  MoveL 660 to (60.77, 126.66, 55.41) mm, rotated rx -112.39 ry 0 rz 153.96 deg; joints [6.851, -47.635, 74.917, -1.241, 56.21, -13.391, 34.019]
  MoveL 661 to (66.75, 124.73, 52.87) mm, rotated rx -111.36 ry 0 rz 151.44 deg; joints [6.623, -47.631, 74.812, -1.242, 56.128, -12.588, 36.717]
  MoveL 662 to (67.07, 124.6, 52.75) mm, rotated rx -111.21 ry 0 rz 151.11 deg; joints [6.599, -47.654, 74.802, -1.244, 56.128, -12.462, 37.079]
  MoveL 663 to (71.33, 123.43, 49.83) mm, rotated rx -110.03 ry 0 rz 149.39 deg; joints [6.337, -47.654, 74.694, -1.241, 56.035, -11.548, 38.999]
  MoveL 664 to (71.29, 123.43, 49.87) mm, rotated rx -109.41 ry 0 rz 148.99 deg; joints [6.253, -47.698, 74.655, -1.242, 56.035, -11.007, 39.475]
  MoveL 665 to (71.98, 123.95, 47.56) mm, rotated rx -108.48 ry 0 rz 148.86 deg; joints [6.046, -47.698, 74.577, -1.235, 55.971, -10.294, 39.744]
  MoveL 666 to (72.34, 124.04, 46.77) mm, rotated rx -108.48 ry 0 rz 148.86 deg; joints [6.02, -47.694, 74.577, -1.235, 55.942, -10.32, 39.769]
  MoveL 667 to (72.46, 124.04, 46.59) mm, rotated rx -108.41 ry 0 rz 148.82 deg; joints [6.003, -47.694, 74.571, -1.234, 55.937, -10.264, 39.82]
  MoveL 668 to (72.72, 124.02, 46.25) mm, rotated rx -108.41 ry 0 rz 148.82 deg; joints [5.992, -47.687, 74.571, -1.234, 55.922, -10.276, 39.827]
  MoveL 669 to (73.92, 123.81, 44.88) mm, rotated rx -107.79 ry 0 rz 148.32 deg; joints [5.859, -47.687, 74.517, -1.226, 55.898, -9.795, 40.405]
  MoveL 670 to (74.21, 123.77, 44.51) mm, rotated rx -107.28 ry 0 rz 148.07 deg; joints [5.775, -47.695, 74.479, -1.22, 55.898, -9.373, 40.699]
  MoveL 671 to (76.55, 125.04, 36.2) mm, rotated rx -104.01 ry 0 rz 147.56 deg; joints [5.033, -47.695, 74.261, -1.159, 55.732, -6.875, 41.585]
  MoveL 672 to (76.56, 125.03, 36.23) mm, rotated rx -103.38 ry 0 rz 147.69 deg; joints [4.944, -47.695, 74.256, -1.152, 55.68, -6.332, 41.508]
  MoveL 673 to (75.15, 126.78, 32.95) mm, rotated rx -102.1 ry 0 rz 148.52 deg; joints [4.651, -47.696, 74.189, -1.119, 55.632, -5.36, 40.791]
  MoveL 674 to (75.18, 126.76, 32.96) mm, rotated rx -101.72 ry 0 rz 149 deg; joints [4.596, -47.646, 74.189, -1.111, 55.58, -5.038, 40.319]
  MoveL 675 to (72.12, 128.85, 31.65) mm, rotated rx -101.21 ry 0 rz 150.43 deg; joints [4.479, -47.646, 74.165, -1.097, 55.564, -4.653, 38.919]
  MoveL 676 to (72.16, 128.83, 31.66) mm, rotated rx -101.17 ry 0 rz 150.93 deg; joints [4.473, -47.583, 74.165, -1.092, 55.536, -4.625, 38.388]
  MoveL 677 to (69.26, 130.27, 32.26) mm, rotated rx -101.4 ry 0 rz 152.18 deg; joints [4.526, -47.583, 74.176, -1.098, 55.543, -4.801, 37.119]
  MoveL 678 to (68.73, 130.53, 32.34) mm, rotated rx -101.43 ry 0 rz 152.35 deg; joints [4.532, -47.591, 74.178, -1.1, 55.545, -4.816, 36.951]
  MoveL 679 to (65.39, 132.13, 32.76) mm, rotated rx -101.64 ry 0 rz 154.01 deg; joints [4.577, -47.56, 74.185, -1.103, 55.545, -4.988, 35.254]
  MoveL 680 to (65.13, 132.23, 32.87) mm, rotated rx -101.68 ry 0 rz 154.12 deg; joints [4.586, -47.561, 74.186, -1.104, 55.546, -5.018, 35.145]
  MoveL 681 to (65.15, 132.23, 32.84) mm, rotated rx -101.9 ry 0 rz 154.47 deg; joints [4.615, -47.509, 74.186, -1.102, 55.544, -5.211, 34.742]
  MoveL 682 to (59.71, 133.3, 38.37) mm, rotated rx -104.07 ry 0 rz 156.58 deg; joints [5.109, -47.509, 74.305, -1.155, 55.627, -6.851, 32.439]
  MoveL 683 to (58.71, 133.57, 39) mm, rotated rx -104.07 ry 0 rz 156.58 deg; joints [5.131, -47.553, 74.305, -1.16, 55.659, -6.827, 32.451]
  MoveL 684 to (58.23, 133.73, 39.16) mm, rotated rx -104.13 ry 0 rz 156.78 deg; joints [5.145, -47.553, 74.308, -1.162, 55.662, -6.875, 32.25]
  MoveL 685 to (57.76, 133.9, 39.27) mm, rotated rx -104.13 ry 0 rz 156.78 deg; joints [5.15, -47.577, 74.308, -1.164, 55.674, -6.87, 32.262]
  MoveL 686 to (52.25, 135.95, 39.92) mm, rotated rx -104.39 ry 0 rz 159.09 deg; joints [5.208, -47.577, 74.324, -1.169, 55.685, -7.065, 29.926]
  MoveL 687 to (51.7, 136.16, 39.92) mm, rotated rx -104.39 ry 0 rz 159.09 deg; joints [5.209, -47.606, 74.324, -1.172, 55.696, -7.063, 29.944]
  MoveL 688 to (50.6, 136.72, 39.43) mm, rotated rx -104.39 ry 0 rz 159.09 deg; joints [5.194, -47.671, 74.325, -1.176, 55.709, -7.076, 29.996]
  MoveL 689 to (50.38, 136.86, 39.24) mm, rotated rx -104.31 ry 0 rz 159.19 deg; joints [5.177, -47.671, 74.32, -1.175, 55.705, -7.018, 29.902]
  MoveL 690 to (49.72, 137.39, 38.2) mm, rotated rx -104.31 ry 0 rz 159.19 deg; joints [5.143, -47.715, 74.316, -1.176, 55.705, -7.052, 29.95]
  MoveL 691 to (49.04, 138.28, 35.81) mm, rotated rx -103.37 ry 0 rz 159.56 deg; joints [4.93, -47.715, 74.262, -1.154, 55.666, -6.341, 29.667]
  MoveL 692 to (48.96, 138.42, 35.38) mm, rotated rx -103.37 ry 0 rz 159.56 deg; joints [4.916, -47.721, 74.258, -1.153, 55.666, -6.356, 29.676]
  MoveL 693 to (49.06, 138.63, 34.37) mm, rotated rx -103.37 ry 0 rz 159.56 deg; joints [4.882, -47.721, 74.251, -1.15, 55.658, -6.392, 29.691]
  MoveL 694 to (49.13, 138.66, 34.16) mm, rotated rx -103.29 ry 0 rz 159.54 deg; joints [4.863, -47.721, 74.246, -1.148, 55.655, -6.331, 29.718]
  MoveL 695 to (49.47, 138.71, 33.44) mm, rotated rx -103.29 ry 0 rz 159.54 deg; joints [4.839, -47.712, 74.246, -1.145, 55.635, -6.356, 29.727]
  MoveL 696 to (50.81, 138.69, 31.45) mm, rotated rx -102.52 ry 0 rz 159.05 deg; joints [4.662, -47.712, 74.207, -1.125, 55.608, -5.771, 30.282]
  MoveL 697 to (51.64, 138.87, 29.25) mm, rotated rx -101.46 ry 0 rz 158.68 deg; joints [4.436, -47.712, 74.148, -1.094, 55.603, -4.949, 30.713]
  MoveL 698 to (51.92, 138.88, 28.69) mm, rotated rx -101.46 ry 0 rz 158.68 deg; joints [4.417, -47.702, 74.148, -1.092, 55.59, -4.969, 30.717]
  MoveL 699 to (52.11, 138.87, 28.42) mm, rotated rx -101.35 ry 0 rz 158.62 deg; joints [4.392, -47.702, 74.143, -1.089, 55.587, -4.89, 30.791]
  MoveL 700 to (52.33, 138.84, 28.13) mm, rotated rx -101.35 ry 0 rz 158.62 deg; joints [4.383, -47.694, 74.143, -1.087, 55.578, -4.9, 30.791]
  MoveL 701 to (53.88, 138.59, 26.37) mm, rotated rx -100.68 ry 0 rz 158.03 deg; joints [4.227, -47.693, 74.116, -1.066, 55.561, -4.391, 31.423]
  MoveL 702 to (53.87, 138.59, 26.41) mm, rotated rx -100.23 ry 0 rz 157.81 deg; joints [4.165, -47.724, 74.108, -1.06, 55.561, -4.012, 31.676]
  MoveL 703 to (54.09, 138.69, 25.45) mm, rotated rx -99.86 ry 0 rz 157.75 deg; joints [4.08, -47.724, 74.095, -1.048, 55.553, -3.735, 31.76]
  MoveL 704 to (54.13, 138.66, 25.45) mm, rotated rx -98.75 ry 0 rz 158.69 deg; joints [3.919, -47.625, 74.095, -1.022, 55.453, -2.799, 30.817]
  MoveL 705 to (46.69, 141.33, 25.56) mm, rotated rx -98.79 ry 0 rz 161.73 deg; joints [3.928, -47.625, 74.096, -1.023, 55.453, -2.829, 27.774]
  MoveL 706 to (46.19, 141.5, 25.51) mm, rotated rx -98.79 ry 0 rz 161.73 deg; joints [3.927, -47.651, 74.096, -1.025, 55.463, -2.83, 27.79]
  MoveL 707 to (45.76, 141.66, 25.42) mm, rotated rx -98.76 ry 0 rz 161.91 deg; joints [3.919, -47.651, 74.094, -1.024, 55.463, -2.803, 27.616]
  MoveL 708 to (44.74, 142.08, 24.9) mm, rotated rx -98.76 ry 0 rz 161.91 deg; joints [3.903, -47.707, 74.094, -1.025, 55.48, -2.819, 27.654]
  MoveL 709 to (41.28, 143.63, 21.8) mm, rotated rx -97.57 ry 0 rz 163.35 deg; joints [3.628, -47.707, 74.061, -0.983, 55.462, -1.926, 26.251]
  MoveL 710 to (40.62, 143.96, 20.83) mm, rotated rx -97.57 ry 0 rz 163.35 deg; joints [3.596, -47.745, 74.061, -0.98, 55.47, -1.959, 26.281]
  MoveL 711 to (40.51, 144.16, 19.63) mm, rotated rx -97.57 ry 0 rz 163.35 deg; joints [3.556, -47.754, 74.058, -0.975, 55.47, -2.002, 26.293]
  MoveL 712 to (40.56, 144.19, 19.26) mm, rotated rx -97.43 ry 0 rz 163.34 deg; joints [3.524, -47.754, 74.055, -0.97, 55.469, -1.897, 26.312]
  MoveL 713 to (40.77, 144.23, 18.53) mm, rotated rx -97.43 ry 0 rz 163.34 deg; joints [3.499, -47.746, 74.055, -0.965, 55.462, -1.924, 26.312]
  MoveL 714 to (42.09, 144.19, 15.65) mm, rotated rx -96.33 ry 0 rz 162.85 deg; joints [3.244, -47.746, 74.035, -0.923, 55.455, -1.102, 26.821]
  MoveL 715 to (42.15, 144.21, 15.29) mm, rotated rx -96.03 ry 0 rz 162.78 deg; joints [3.189, -47.754, 74.033, -0.915, 55.455, -0.864, 26.904]
  MoveL 716 to (43.13, 144.27, 11.53) mm, rotated rx -94.6 ry 0 rz 162.43 deg; joints [2.857, -47.755, 74.02, -0.858, 55.455, 0.205, 27.261]
  MoveL 717 to (43.15, 144.26, 11.55) mm, rotated rx -93.63 ry 0 rz 162.78 deg; joints [2.716, -47.713, 74.02, -0.831, 55.435, 1.024, 26.893]
  MoveL 718 to (37.84, 146.01, 7.35) mm, rotated rx -92.03 ry 0 rz 164.9 deg; joints [2.344, -47.713, 74.024, -0.764, 55.452, 2.216, 24.742]
  MoveL 719 to (37.83, 146.02, 7.37) mm, rotated rx -91.85 ry 0 rz 165.55 deg; joints [2.317, -47.629, 74.024, -0.755, 55.419, 2.366, 24.038]
  MoveL 720 to (29.7, 147.83, 8.53) mm, rotated rx -92.3 ry 0 rz 168.77 deg; joints [2.421, -47.626, 74.024, -0.774, 55.405, 2.032, 20.832]
  MoveL 721 to (28.41, 148.09, 8.36) mm, rotated rx -92.3 ry 0 rz 168.77 deg; joints [2.416, -47.69, 74.024, -0.776, 55.433, 2.027, 20.868]
  MoveL 722 to (28.01, 148.18, 8.19) mm, rotated rx -92.23 ry 0 rz 168.93 deg; joints [2.401, -47.69, 74.025, -0.773, 55.433, 2.076, 20.712]
  MoveL 723 to (25.31, 148.72, 6.82) mm, rotated rx -91.74 ry 0 rz 169.92 deg; joints [2.283, -47.692, 74.025, -0.752, 55.451, 2.443, 19.703]
  MoveL 724 to (25.34, 148.72, 6.79) mm, rotated rx -91.84 ry 0 rz 170.93 deg; joints [2.295, -47.562, 74.025, -0.748, 55.394, 2.352, 18.619]
  MoveL 725 to (23.1, 148.99, 8.62) mm, rotated rx -92.54 ry 0 rz 171.79 deg; joints [2.457, -47.562, 74.02, -0.778, 55.384, 1.832, 17.778]
  MoveL 726 to (22.86, 149.01, 8.97) mm, rotated rx -92.78 ry 0 rz 171.99 deg; joints [2.503, -47.549, 74.02, -0.785, 55.374, 1.64, 17.57]
  MoveL 727 to (20.3, 149.18, 11.9) mm, rotated rx -93.9 ry 0 rz 172.97 deg; joints [2.763, -47.548, 74.02, -0.831, 55.365, 0.807, 16.605]
  MoveL 728 to (19.26, 149.26, 12.61) mm, rotated rx -93.9 ry 0 rz 172.97 deg; joints [2.787, -47.599, 74.02, -0.838, 55.385, 0.834, 16.635]
  MoveL 729 to (18.7, 149.31, 12.81) mm, rotated rx -93.97 ry 0 rz 173.18 deg; joints [2.805, -47.598, 74.02, -0.841, 55.385, 0.777, 16.421]
  MoveL 730 to (18.28, 149.35, 12.92) mm, rotated rx -93.97 ry 0 rz 173.18 deg; joints [2.809, -47.619, 74.02, -0.843, 55.394, 0.782, 16.433]
  MoveL 731 to (13.22, 149.81, 13.78) mm, rotated rx -94.38 ry 0 rz 175.37 deg; joints [2.897, -47.584, 74.02, -0.856, 55.383, 0.467, 14.224]
  MoveL 732 to (10.64, 149.89, 15.02) mm, rotated rx -94.86 ry 0 rz 176.35 deg; joints [3.006, -47.583, 74.023, -0.875, 55.384, 0.114, 13.236]
  MoveL 733 to (9.93, 149.91, 15.35) mm, rotated rx -94.92 ry 0 rz 176.45 deg; joints [3.026, -47.604, 74.023, -0.879, 55.394, 0.075, 13.148]
  MoveL 734 to (7.35, 149.99, 16.03) mm, rotated rx -95.18 ry 0 rz 177.44 deg; joints [3.087, -47.604, 74.026, -0.889, 55.394, -0.119, 12.161]
  MoveL 735 to (8.24, 169.89, 17.83) mm, rotated rx -95.18 ry 0 rz 177.44 deg; joints [3.116, -46.976, 72.196, -1.011, 55.394, -0.037, 13.368]
  Set speed (1000.0 mm/s)
  MoveL 736 to (4.59, 170.21, 15.87) mm, rotated rx -94.56 ry 0 rz 178.8 deg; joints [2.963, -46.964, 72.196, -0.981, 55.377, 0.408, 12.008]
  Set speed (5.0 mm/s)
  MoveL 737 to (4.17, 150.28, 14.28) mm, rotated rx -94.56 ry 0 rz 178.8 deg; joints [2.94, -47.591, 74.026, -0.864, 55.377, 0.334, 10.801]
  Set speed (16.7 mm/s)
  MoveL 738 to (2.77, 150.26, 14.91) mm, rotated rx -94.8 ry 0 rz 179.33 deg; joints [2.995, -47.591, 74.027, -0.874, 55.377, 0.156, 10.266]
  MoveL 739 to (1.49, 150.25, 15.12) mm, rotated rx -94.8 ry 0 rz 179.33 deg; joints [3.003, -47.653, 74.027, -0.878, 55.403, 0.165, 10.302]
  MoveL 740 to (1.28, 150.26, 15.1) mm, rotated rx -94.79 ry 0 rz 179.42 deg; joints [3.001, -47.653, 74.027, -0.878, 55.403, 0.172, 10.222]
  MoveL 741 to (0.58, 150.28, 14.92) mm, rotated rx -94.79 ry 0 rz 179.42 deg; joints [2.996, -47.687, 74.027, -0.879, 55.417, 0.166, 10.242]
  MoveL 742 to (-0.95, 150.34, 14.29) mm, rotated rx -94.55 ry 0 rz 180 deg; joints [2.94, -47.687, 74.026, -0.869, 55.417, 0.344, 9.659]
  MoveL 743 to (-2.76, 150.39, 13.54) mm, rotated rx -94.27 ry 0 rz -179.31 deg; joints [2.874, -47.688, 74.024, -0.858, 55.417, 0.558, 8.969]
  MoveL 744 to (-3.05, 150.39, 13.4) mm, rotated rx -94.27 ry 0 rz -179.31 deg; joints [2.87, -47.702, 74.024, -0.858, 55.423, 0.554, 8.978]
  MoveL 745 to (-3.44, 150.4, 13.18) mm, rotated rx -94.18 ry 0 rz -179.16 deg; joints [2.85, -47.702, 74.024, -0.854, 55.423, 0.617, 8.829]
  MoveL 746 to (-5.89, 150.44, 11.76) mm, rotated rx -93.65 ry 0 rz -178.24 deg; joints [2.725, -47.705, 74.024, -0.833, 55.423, 1.017, 7.906]
  MoveL 747 to (-5.83, 150.44, 11.77) mm, rotated rx -93.52 ry 0 rz -177.74 deg; joints [2.706, -47.638, 74.024, -0.826, 55.395, 1.122, 7.365]
  MoveL 748 to (-8.98, 150.28, 11.92) mm, rotated rx -93.58 ry 0 rz -176.54 deg; joints [2.719, -47.638, 74.024, -0.828, 55.395, 1.079, 6.165]
  MoveL 749 to (-9.52, 150.25, 11.88) mm, rotated rx -93.58 ry 0 rz -176.54 deg; joints [2.718, -47.664, 74.024, -0.83, 55.406, 1.079, 6.181]
  MoveL 750 to (-10.04, 150.22, 11.79) mm, rotated rx -93.54 ry 0 rz -176.34 deg; joints [2.71, -47.664, 74.024, -0.828, 55.406, 1.105, 5.981]
  MoveL 751 to (-10.45, 150.2, 11.69) mm, rotated rx -93.54 ry 0 rz -176.34 deg; joints [2.707, -47.684, 74.024, -0.829, 55.414, 1.102, 5.993]
  MoveL 752 to (-13.43, 150.04, 10.65) mm, rotated rx -93.15 ry 0 rz -175.2 deg; joints [2.615, -47.684, 74.024, -0.812, 55.418, 1.397, 4.851]
  MoveL 753 to (-13.42, 150.04, 10.63) mm, rotated rx -93.18 ry 0 rz -174.48 deg; joints [2.618, -47.592, 74.024, -0.808, 55.379, 1.365, 4.081]
  MoveL 754 to (-16.19, 149.67, 11.96) mm, rotated rx -93.68 ry 0 rz -173.42 deg; joints [2.735, -47.592, 74.024, -0.829, 55.375, 0.99, 3.023]
  MoveL 755 to (-16.97, 149.57, 12.18) mm, rotated rx -93.68 ry 0 rz -173.42 deg; joints [2.743, -47.63, 74.024, -0.832, 55.391, 0.999, 3.046]
  MoveL 756 to (-17.85, 149.46, 12.28) mm, rotated rx -93.72 ry 0 rz -173.08 deg; joints [2.752, -47.63, 74.024, -0.834, 55.391, 0.97, 2.709]
  MoveL 757 to (-19.05, 149.32, 12.12) mm, rotated rx -93.72 ry 0 rz -173.08 deg; joints [2.748, -47.689, 74.024, -0.836, 55.416, 0.966, 2.743]
  MoveL 758 to (-23.23, 148.85, 10.44) mm, rotated rx -93.08 ry 0 rz -171.48 deg; joints [2.599, -47.689, 74.024, -0.809, 55.42, 1.444, 1.136]
  MoveL 759 to (-23.2, 148.86, 10.45) mm, rotated rx -93.07 ry 0 rz -170.84 deg; joints [2.596, -47.606, 74.024, -0.805, 55.385, 1.454, 0.451]
  MoveL 760 to (-25.12, 148.5, 11.09) mm, rotated rx -93.31 ry 0 rz -170.1 deg; joints [2.652, -47.606, 74.024, -0.815, 55.383, 1.273, -0.288]
  MoveL 761 to (-26.31, 148.29, 11.17) mm, rotated rx -93.2 ry 0 rz -170.09 deg; joints [2.64, -47.663, 74.024, -0.816, 55.407, 1.372, -0.273]
  MoveL 762 to (-27.06, 148.18, 10.9) mm, rotated rx -93.13 ry 0 rz -170.07 deg; joints [2.621, -47.698, 74.024, -0.814, 55.423, 1.425, -0.264]
  MoveL 763 to (-27.67, 148.1, 10.44) mm, rotated rx -93.06 ry 0 rz -170.06 deg; joints [2.595, -47.726, 74.024, -0.81, 55.436, 1.468, -0.261]
  MoveL 764 to (-28.2, 148.05, 9.57) mm, rotated rx -92.96 ry 0 rz -170.05 deg; joints [2.553, -47.75, 74.024, -0.804, 55.449, 1.516, -0.264]
  MoveL 765 to (-28.34, 148.09, 8.55) mm, rotated rx -92.87 ry 0 rz -170.04 deg; joints [2.506, -47.754, 74.024, -0.795, 55.454, 1.559, -0.28]
  MoveL 766 to (-29.06, 148.04, 6.92) mm, rotated rx -92.25 ry 0 rz -169.76 deg; joints [2.361, -47.755, 74.027, -0.769, 55.461, 2.023, -0.563]
  MoveL 767 to (-28.94, 148.05, 7.15) mm, rotated rx -92.25 ry 0 rz -169.76 deg; joints [2.369, -47.749, 74.027, -0.77, 55.458, 2.031, -0.566]
  MoveL 768 to (-29.05, 148.04, 6.96) mm, rotated rx -92.17 ry 0 rz -169.72 deg; joints [2.352, -47.749, 74.027, -0.767, 55.459, 2.085, -0.608]
  MoveL 769 to (-29.31, 148.01, 6.46) mm, rotated rx -92.03 ry 0 rz -169.65 deg; joints [2.314, -47.751, 74.027, -0.76, 55.465, 2.19, -0.686]
  MoveL 770 to (-29.27, 148.01, 6.49) mm, rotated rx -91.56 ry 0 rz -169.1 deg; joints [2.246, -47.676, 74.027, -0.744, 55.443, 2.584, -1.29]
  MoveL 771 to (-31.93, 147.5, 5.64) mm, rotated rx -91.23 ry 0 rz -168.07 deg; joints [2.17, -47.676, 74.03, -0.73, 55.448, 2.824, -2.327]
  MoveL 772 to (-32.39, 147.41, 5.43) mm, rotated rx -91.23 ry 0 rz -168.07 deg; joints [2.164, -47.699, 74.03, -0.73, 55.459, 2.817, -2.315]
  MoveL 773 to (-32.76, 147.33, 5.22) mm, rotated rx -91.15 ry 0 rz -167.93 deg; joints [2.145, -47.699, 74.032, -0.727, 55.46, 2.877, -2.462]
  MoveL 774 to (-33.25, 147.24, 4.86) mm, rotated rx -91.15 ry 0 rz -167.93 deg; joints [2.134, -47.722, 74.032, -0.725, 55.472, 2.864, -2.45]
  MoveL 775 to (-36.36, 146.57, 1.84) mm, rotated rx -90.01 ry 0 rz -166.72 deg; joints [1.867, -47.722, 74.049, -0.676, 55.497, 3.717, -3.706]
  MoveL 776 to (-36.4, 146.55, 1.78) mm, rotated rx -89.81 ry 0 rz -166.43 deg; joints [1.835, -47.684, 74.049, -0.668, 55.491, 3.884, -4.024]
  MoveL 777 to (-41.32, 145.25, -0.45) mm, rotated rx -88.96 ry 0 rz -164.5 deg; joints [1.638, -47.685, 74.067, -0.631, 55.513, 4.515, -5.996]
  MoveL 778 to (-41.25, 145.28, -0.43) mm, rotated rx -88.89 ry 0 rz -164.17 deg; joints [1.628, -47.637, 74.067, -0.627, 55.497, 4.575, -6.361]
  MoveL 779 to (-45.56, 143.99, -0.15) mm, rotated rx -89 ry 0 rz -162.38 deg; joints [1.653, -47.63, 74.067, -0.632, 55.485, 4.493, -8.142]
  MoveL 780 to (-46.02, 143.84, -0.16) mm, rotated rx -89 ry 0 rz -162.38 deg; joints [1.653, -47.653, 74.067, -0.633, 55.495, 4.493, -8.128]
  MoveL 781 to (-47.03, 143.51, -0.3) mm, rotated rx -88.95 ry 0 rz -161.98 deg; joints [1.641, -47.653, 74.069, -0.631, 55.496, 4.532, -8.537]
  MoveL 782 to (-47.66, 143.3, -0.48) mm, rotated rx -88.95 ry 0 rz -161.98 deg; joints [1.635, -47.685, 74.069, -0.631, 55.511, 4.527, -8.52]
  MoveL 783 to (-54.7, 140.72, -3.71) mm, rotated rx -87.72 ry 0 rz -159.13 deg; joints [1.35, -47.685, 74.103, -0.577, 55.55, 5.44, -11.441]
  MoveL 784 to (-54.97, 140.61, -3.86) mm, rotated rx -87.72 ry 0 rz -159.13 deg; joints [1.345, -47.698, 74.103, -0.577, 55.558, 5.435, -11.435]
  MoveL 785 to (-55.36, 140.45, -4.11) mm, rotated rx -87.62 ry 0 rz -158.97 deg; joints [1.323, -47.698, 74.106, -0.572, 55.561, 5.507, -11.604]
  MoveL 786 to (-55.65, 140.33, -4.33) mm, rotated rx -87.62 ry 0 rz -158.97 deg; joints [1.316, -47.712, 74.106, -0.571, 55.57, 5.499, -11.599]
  MoveL 787 to (-58.19, 139.2, -6.59) mm, rotated rx -86.76 ry 0 rz -157.91 deg; joints [1.116, -47.712, 74.136, -0.534, 55.601, 6.141, -12.718]
  MoveL 788 to (-58.87, 138.86, -7.66) mm, rotated rx -86.76 ry 0 rz -157.91 deg; joints [1.081, -47.743, 74.136, -0.528, 55.632, 6.102, -12.717]
  MoveL 789 to (-58.95, 138.82, -7.88) mm, rotated rx -86.68 ry 0 rz -157.88 deg; joints [1.061, -47.744, 74.139, -0.524, 55.636, 6.166, -12.756]
  MoveL 790 to (-59.04, 138.76, -8.27) mm, rotated rx -86.68 ry 0 rz -157.88 deg; joints [1.048, -47.748, 74.14, -0.522, 55.642, 6.152, -12.76]
  MoveL 791 to (-59.34, 138.5, -10.19) mm, rotated rx -85.95 ry 0 rz -157.74 deg; joints [0.879, -47.748, 74.17, -0.49, 55.673, 6.695, -12.965]
  MoveL 792 to (-59.48, 138.42, -10.44) mm, rotated rx -85.61 ry 0 rz -157.6 deg; joints [0.822, -47.741, 74.185, -0.479, 55.673, 6.968, -13.13]
  MoveL 793 to (-61.44, 137.13, -15.06) mm, rotated rx -83.86 ry 0 rz -156.72 deg; joints [0.415, -47.741, 74.272, -0.404, 55.76, 8.281, -14.185]
  MoveL 794 to (-61.42, 137.14, -15.03) mm, rotated rx -83.46 ry 0 rz -156.34 deg; joints [0.358, -47.687, 74.281, -0.392, 55.76, 8.616, -14.629]
  MoveL 795 to (-63.42, 136.09, -16.28) mm, rotated rx -82.98 ry 0 rz -155.48 deg; joints [0.248, -47.687, 74.308, -0.373, 55.787, 8.972, -15.545]
  MoveL 796 to (-63.67, 135.95, -16.43) mm, rotated rx -82.92 ry 0 rz -155.36 deg; joints [0.234, -47.687, 74.312, -0.37, 55.788, 9.019, -15.667]
  MoveL 797 to (-65.55, 134.9, -17.63) mm, rotated rx -82.47 ry 0 rz -154.55 deg; joints [0.129, -47.687, 74.338, -0.351, 55.818, 9.356, -16.532]
  MoveL 798 to (-65.54, 134.91, -17.62) mm, rotated rx -82.36 ry 0 rz -154.01 deg; joints [0.113, -47.612, 74.338, -0.347, 55.802, 9.45, -17.132]
  MoveL 799 to (-66.71, 134.35, -17.51) mm, rotated rx -82.4 ry 0 rz -153.51 deg; joints [0.122, -47.612, 74.336, -0.349, 55.799, 9.42, -17.624]
  MoveL 800 to (-67.08, 134.17, -17.51) mm, rotated rx -82.4 ry 0 rz -153.51 deg; joints [0.123, -47.633, 74.336, -0.349, 55.807, 9.42, -17.611]
  MoveL 801 to (-67.61, 133.9, -17.56) mm, rotated rx -82.38 ry 0 rz -153.29 deg; joints [0.118, -47.633, 74.337, -0.348, 55.808, 9.434, -17.837]
  MoveL 802 to (-67.99, 133.69, -17.63) mm, rotated rx -82.38 ry 0 rz -153.29 deg; joints [0.116, -47.654, 74.337, -0.348, 55.818, 9.431, -17.826]
  MoveL 803 to (-71.95, 131.43, -18.84) mm, rotated rx -81.92 ry 0 rz -151.55 deg; joints [0.01, -47.654, 74.366, -0.329, 55.846, 9.777, -19.625]
  MoveL 804 to (-72.27, 131.25, -18.94) mm, rotated rx -81.88 ry 0 rz -151.42 deg; joints [0.001, -47.654, 74.367, -0.328, 55.852, 9.803, -19.759]
  MoveL 805 to (-74.67, 129.78, -19.68) mm, rotated rx -81.6 ry 0 rz -150.33 deg; joints [-0.064, -47.654, 74.387, -0.317, 55.866, 10.017, -20.886]
  MoveL 806 to (-75.35, 129.33, -20.05) mm, rotated rx -81.6 ry 0 rz -150.33 deg; joints [-0.077, -47.69, 74.387, -0.315, 55.89, 10.004, -20.874]
  MoveL 807 to (-75.55, 129.19, -20.23) mm, rotated rx -81.53 ry 0 rz -150.23 deg; joints [-0.092, -47.69, 74.392, -0.312, 55.894, 10.054, -20.977]
  MoveL 808 to (-75.96, 128.88, -20.7) mm, rotated rx -81.53 ry 0 rz -150.23 deg; joints [-0.108, -47.71, 74.392, -0.31, 55.916, 10.037, -20.979]
  MoveL 809 to (-76.86, 128.09, -22.15) mm, rotated rx -80.97 ry 0 rz -149.79 deg; joints [-0.236, -47.71, 74.43, -0.288, 55.953, 10.454, -21.503]
  MoveL 810 to (-76.83, 128.11, -22.14) mm, rotated rx -80.62 ry 0 rz -149.03 deg; joints [-0.286, -47.598, 74.432, -0.277, 55.953, 10.75, -22.374]
  MoveL 811 to (-78.76, 126.95, -22.09) mm, rotated rx -80.64 ry 0 rz -148.16 deg; joints [-0.282, -47.598, 74.431, -0.278, 55.952, 10.737, -23.238]
  MoveL 812 to (-79.07, 126.75, -22.11) mm, rotated rx -80.64 ry 0 rz -148.16 deg; joints [-0.282, -47.616, 74.431, -0.278, 55.959, 10.736, -23.227]
  MoveL 813 to (-79.56, 126.43, -22.19) mm, rotated rx -80.61 ry 0 rz -147.94 deg; joints [-0.289, -47.616, 74.433, -0.277, 55.961, 10.757, -23.456]
  MoveL 814 to (-83.97, 123.36, -23.2) mm, rotated rx -80.21 ry 0 rz -145.74 deg; joints [-0.38, -47.611, 74.475, -0.262, 55.96, 11.058, -25.702]
  MoveL 815 to (-84.11, 123.27, -23.2) mm, rotated rx -80.21 ry 0 rz -145.68 deg; joints [-0.38, -47.611, 74.475, -0.262, 55.96, 11.057, -25.766]
  MoveL 816 to (-86.01, 122, -22.94) mm, rotated rx -80.32 ry 0 rz -144.71 deg; joints [-0.356, -47.607, 74.474, -0.266, 55.936, 10.978, -26.71]
  MoveL 817 to (-86.54, 121.62, -22.95) mm, rotated rx -80.32 ry 0 rz -144.71 deg; joints [-0.356, -47.639, 74.475, -0.266, 55.948, 10.977, -26.689]
  MoveL 818 to (-87.53, 120.87, -23.14) mm, rotated rx -80.25 ry 0 rz -144.23 deg; joints [-0.372, -47.639, 74.48, -0.264, 55.953, 11.031, -27.177]
  MoveL 819 to (-88.19, 120.34, -23.43) mm, rotated rx -80.25 ry 0 rz -144.23 deg; joints [-0.382, -47.678, 74.48, -0.263, 55.977, 11.021, -27.162]
  MoveL 820 to (-91.78, 117.05, -26.1) mm, rotated rx -79.22 ry 0 rz -142.37 deg; joints [-0.618, -47.678, 74.559, -0.224, 56.054, 11.794, -29.18]
  MoveL 821 to (-94.95, 113.9, -28.59) mm, rotated rx -78.17 ry 0 rz -140.41 deg; joints [-0.85, -47.678, 74.674, -0.187, 56.07, 12.597, -31.272]
  MoveL 822 to (-97.63, 111.54, -28.88) mm, rotated rx -78.03 ry 0 rz -138.89 deg; joints [-0.879, -47.662, 74.687, -0.183, 56.07, 12.701, -32.826]
  MoveL 823 to (-98.35, 110.83, -29.18) mm, rotated rx -78.03 ry 0 rz -138.89 deg; joints [-0.889, -47.709, 74.687, -0.181, 56.097, 12.691, -32.807]
  MoveL 824 to (-98.66, 110.49, -29.43) mm, rotated rx -77.93 ry 0 rz -138.71 deg; joints [-0.911, -47.709, 74.695, -0.178, 56.105, 12.764, -33]
  MoveL 825 to (-98.92, 110.18, -29.71) mm, rotated rx -77.93 ry 0 rz -138.71 deg; joints [-0.92, -47.725, 74.695, -0.177, 56.121, 12.754, -33]
  MoveL 826 to (-99.3, 109.59, -30.59) mm, rotated rx -77.93 ry 0 rz -138.71 deg; joints [-0.949, -47.747, 74.695, -0.172, 56.162, 12.722, -33.02]
  MoveL 827 to (-100.29, 106.94, -36.23) mm, rotated rx -75.74 ry 0 rz -137.74 deg; joints [-1.447, -47.748, 74.899, -0.099, 56.361, 14.379, -34.396]
  MoveL 828 to (-100.26, 106.61, -37.26) mm, rotated rx -75.74 ry 0 rz -137.74 deg; joints [-1.481, -47.748, 74.904, -0.095, 56.395, 14.343, -34.436]
  MoveL 829 to (-99.99, 106.37, -38.65) mm, rotated rx -75.2 ry 0 rz -137.75 deg; joints [-1.604, -47.748, 74.96, -0.078, 56.448, 14.755, -34.527]
  MoveL 830 to (-99.85, 106.32, -39.13) mm, rotated rx -75.2 ry 0 rz -137.75 deg; joints [-1.62, -47.748, 74.97, -0.076, 56.449, 14.738, -34.538]
  MoveL 831 to (-99.3, 106.47, -40.12) mm, rotated rx -75.2 ry 0 rz -137.75 deg; joints [-1.653, -47.727, 74.989, -0.072, 56.449, 14.703, -34.579]
  MoveL 832 to (-95.86, 107.97, -44.27) mm, rotated rx -73.55 ry 0 rz -139.17 deg; joints [-2.022, -47.727, 75.167, -0.027, 56.625, 15.957, -33.519]
  MoveL 833 to (-92.33, 109.27, -48.4) mm, rotated rx -71.91 ry 0 rz -140.58 deg; joints [-2.388, -47.727, 75.357, 0.011, 56.818, 17.217, -32.489]
  MoveL 834 to (-90.69, 109.58, -50.75) mm, rotated rx -70.84 ry 0 rz -141.26 deg; joints [-2.614, -47.727, 75.471, 0.031, 56.967, 18.047, -32.076]
  MoveL 835 to (-90.15, 109.74, -51.35) mm, rotated rx -70.54 ry 0 rz -141.5 deg; joints [-2.676, -47.727, 75.502, 0.036, 57.012, 18.285, -31.907]
  MoveL 836 to (-87.46, 109.87, -55.55) mm, rotated rx -68.83 ry 0 rz -142.4 deg; joints [-3.05, -47.727, 75.725, 0.062, 57.245, 19.606, -31.468]
  MoveL 837 to (-87.46, 109.88, -55.52) mm, rotated rx -68.22 ry 0 rz -142.48 deg; joints [-3.132, -47.727, 75.767, 0.066, 57.319, 20.135, -31.504]
  MoveL 838 to (-87.35, 108.92, -57.57) mm, rotated rx -67.38 ry 0 rz -142.27 deg; joints [-3.314, -47.727, 75.882, 0.075, 57.442, 20.786, -31.946]
  MoveL 839 to (-87.26, 108.71, -58.1) mm, rotated rx -67.38 ry 0 rz -142.27 deg; joints [-3.332, -47.727, 75.891, 0.075, 57.461, 20.768, -31.973]
  MoveL 840 to (-87.16, 108.58, -58.48) mm, rotated rx -67.22 ry 0 rz -142.27 deg; joints [-3.366, -47.727, 75.913, 0.077, 57.485, 20.892, -32.018]
  MoveL 841 to (-87.08, 108.51, -58.74) mm, rotated rx -67.22 ry 0 rz -142.27 deg; joints [-3.375, -47.727, 75.92, 0.077, 57.489, 20.883, -32.029]
  MoveL 842 to (-85.74, 107.56, -62.34) mm, rotated rx -65.73 ry 0 rz -142.48 deg; joints [-3.696, -47.727, 76.137, 0.085, 57.725, 22.05, -32.279]
  MoveL 843 to (-85.5, 107.47, -62.83) mm, rotated rx -65.73 ry 0 rz -142.48 deg; joints [-3.712, -47.727, 76.154, 0.086, 57.725, 22.034, -32.297]
  MoveL 844 to (-85.36, 107.44, -63.08) mm, rotated rx -65.63 ry 0 rz -142.52 deg; joints [-3.734, -47.727, 76.17, 0.086, 57.742, 22.115, -32.289]
  MoveL 845 to (-85.15, 107.42, -63.39) mm, rotated rx -65.63 ry 0 rz -142.52 deg; joints [-3.745, -47.723, 76.181, 0.086, 57.742, 22.105, -32.304]
  MoveL 846 to (-84.01, 107.4, -64.91) mm, rotated rx -64.99 ry 0 rz -142.89 deg; joints [-3.881, -47.723, 76.277, 0.087, 57.851, 22.609, -32.133]
  MoveL 847 to (-84.04, 107.41, -64.86) mm, rotated rx -64.47 ry 0 rz -143.01 deg; joints [-3.948, -47.723, 76.311, 0.086, 57.932, 23.059, -32.133]
  MoveL 848 to (-83.77, 106.83, -66.17) mm, rotated rx -63.92 ry 0 rz -142.95 deg; joints [-4.065, -47.735, 76.408, 0.086, 58.007, 23.492, -32.351]
  MoveL 849 to (-83.49, 106.57, -66.94) mm, rotated rx -63.92 ry 0 rz -142.95 deg; joints [-4.091, -47.736, 76.431, 0.085, 58.022, 23.467, -32.388]
  MoveL 850 to (-83.37, 106.52, -67.16) mm, rotated rx -63.82 ry 0 rz -142.98 deg; joints [-4.111, -47.739, 76.449, 0.085, 58.034, 23.542, -32.388]
  MoveL 851 to (-82.97, 106.45, -67.77) mm, rotated rx -63.82 ry 0 rz -142.98 deg; joints [-4.131, -47.732, 76.472, 0.085, 58.034, 23.522, -32.418]
  MoveL 852 to (-80.87, 106.44, -70.28) mm, rotated rx -62.75 ry 0 rz -143.69 deg; joints [-4.357, -47.732, 76.643, 0.078, 58.232, 24.374, -32.068]
  MoveL 853 to (-80.38, 106.41, -70.87) mm, rotated rx -62.47 ry 0 rz -143.87 deg; joints [-4.413, -47.732, 76.685, 0.076, 58.287, 24.596, -31.99]
  MoveL 854 to (-80.11, 106.42, -71.17) mm, rotated rx -62.47 ry 0 rz -143.87 deg; joints [-4.423, -47.725, 76.697, 0.075, 58.287, 24.586, -32.009]
  MoveL 855 to (-75.14, 106.77, -75.91) mm, rotated rx -60.41 ry 0 rz -145.73 deg; joints [-4.85, -47.725, 77.041, 0.047, 58.702, 26.239, -30.913]
  MoveL 856 to (-74.77, 106.81, -76.21) mm, rotated rx -60.41 ry 0 rz -145.73 deg; joints [-4.86, -47.711, 77.054, 0.046, 58.702, 26.229, -30.94]
  MoveL 857 to (-73.82, 107.15, -76.66) mm, rotated rx -60.41 ry 0 rz -145.73 deg; joints [-4.875, -47.665, 77.073, 0.042, 58.702, 26.217, -31.006]
  MoveL 858 to (-73.35, 107.38, -76.79) mm, rotated rx -60.35 ry 0 rz -145.96 deg; joints [-4.887, -47.665, 77.083, 0.041, 58.714, 26.261, -30.796]
  MoveL 859 to (-73.05, 107.55, -76.85) mm, rotated rx -60.35 ry 0 rz -145.96 deg; joints [-4.888, -47.647, 77.085, 0.04, 58.714, 26.26, -30.816]
  MoveL 860 to (-68.65, 110, -77.42) mm, rotated rx -60.1 ry 0 rz -148.18 deg; joints [-4.94, -47.647, 77.128, 0.035, 58.768, 26.462, -28.695]
  MoveL 861 to (-66.58, 110.63, -78.32) mm, rotated rx -59.61 ry 0 rz -149.45 deg; joints [-5.033, -47.647, 77.167, 0.022, 58.946, 26.868, -27.637]
  MoveL 862 to (-65.98, 110.84, -78.54) mm, rotated rx -59.42 ry 0 rz -149.91 deg; joints [-5.064, -47.647, 77.173, 0.018, 59.02, 27.031, -27.263]
  MoveL 863 to (-60.49, 111.53, -81.89) mm, rotated rx -57.91 ry 0 rz -152.21 deg; joints [-5.368, -47.647, 77.44, -0.021, 59.364, 28.252, -25.566]
  MoveL 864 to (-60.48, 111.53, -81.9) mm, rotated rx -57.06 ry 0 rz -152.65 deg; joints [-5.474, -47.647, 77.486, -0.041, 59.587, 29.008, -25.397]
  MoveL 865 to (-59.61, 108.8, -86.12) mm, rotated rx -55.14 ry 0 rz -152.43 deg; joints [-5.862, -47.915, 78.097, -0.067, 59.588, 30.558, -25.966]
  MoveL 866 to (-59.48, 108.55, -86.53) mm, rotated rx -55.14 ry 0 rz -152.43 deg; joints [-5.876, -47.925, 78.12, -0.068, 59.588, 30.544, -25.979]
  MoveL 867 to (-58.88, 108.18, -87.39) mm, rotated rx -55.14 ry 0 rz -152.43 deg; joints [-5.906, -47.926, 78.169, -0.072, 59.588, 30.516, -26.028]
  MoveL 868 to (-58.7, 108.13, -87.58) mm, rotated rx -55.05 ry 0 rz -152.49 deg; joints [-5.923, -47.926, 78.185, -0.075, 59.611, 30.588, -26.001]
  MoveL 869 to (-58.54, 108.09, -87.73) mm, rotated rx -55.05 ry 0 rz -152.49 deg; joints [-5.928, -47.923, 78.194, -0.076, 59.611, 30.583, -26.013]
  MoveL 870 to (-56.56, 107.72, -89.47) mm, rotated rx -54.23 ry 0 rz -153.24 deg; joints [-6.087, -47.923, 78.349, -0.11, 59.828, 31.259, -25.639]
  MoveL 871 to (-54.65, 107.13, -91.35) mm, rotated rx -53.27 ry 0 rz -153.99 deg; joints [-6.267, -47.924, 78.522, -0.153, 60.097, 32.061, -25.338]
  MoveL 872 to (-54.31, 107.05, -91.64) mm, rotated rx -53.27 ry 0 rz -153.99 deg; joints [-6.277, -47.916, 78.541, -0.156, 60.097, 32.052, -25.364]
  MoveL 873 to (-53.99, 107.01, -91.88) mm, rotated rx -53.16 ry 0 rz -154.11 deg; joints [-6.299, -47.917, 78.563, -0.161, 60.129, 32.147, -25.289]
  MoveL 874 to (-51.7, 106.68, -93.55) mm, rotated rx -52.36 ry 0 rz -155.04 deg; joints [-6.452, -47.918, 78.721, -0.202, 60.357, 32.815, -24.755]
  MoveL 875 to (-51.72, 106.71, -93.51) mm, rotated rx -51.87 ry 0 rz -155.33 deg; joints [-6.508, -47.918, 78.746, -0.22, 60.508, 33.259, -24.633]
  MoveL 876 to (-51.32, 106.17, -94.35) mm, rotated rx -51.46 ry 0 rz -155.41 deg; joints [-6.586, -47.983, 78.888, -0.23, 60.508, 33.59, -24.637]
  MoveL 877 to (-51.01, 105.9, -94.82) mm, rotated rx -51.46 ry 0 rz -155.41 deg; joints [-6.603, -47.988, 78.918, -0.233, 60.508, 33.575, -24.663]
  MoveL 878 to (-50.61, 105.7, -95.25) mm, rotated rx -51.43 ry 0 rz -155.42 deg; joints [-6.622, -47.991, 78.955, -0.237, 60.508, 33.592, -24.679]
  MoveL 879 to (-49.82, 105.45, -95.95) mm, rotated rx -51.09 ry 0 rz -155.73 deg; joints [-6.686, -47.994, 79.026, -0.256, 60.607, 33.881, -24.546]
  MoveL 880 to (-49.34, 104.96, -96.73) mm, rotated rx -50.4 ry 0 rz -156.02 deg; joints [-6.797, -48.108, 79.229, -0.269, 60.609, 34.465, -24.345]
  MoveL 881 to (-49.02, 104.73, -97.14) mm, rotated rx -50.4 ry 0 rz -156.02 deg; joints [-6.811, -48.11, 79.257, -0.273, 60.609, 34.453, -24.371]
  MoveL 882 to (-48.71, 104.57, -97.47) mm, rotated rx -50.23 ry 0 rz -156.13 deg; joints [-6.843, -48.137, 79.316, -0.277, 60.611, 34.588, -24.294]
  MoveL 883 to (-48.28, 104.42, -97.85) mm, rotated rx -50.23 ry 0 rz -156.13 deg; joints [-6.856, -48.131, 79.342, -0.281, 60.611, 34.577, -24.327]
  MoveL 884 to (-43.98, 103.32, -100.99) mm, rotated rx -48.64 ry 0 rz -157.91 deg; joints [-7.157, -48.408, 79.924, -0.327, 60.611, 35.893, -22.851]
  MoveL 885 to (-43.55, 103.24, -101.26) mm, rotated rx -48.64 ry 0 rz -157.91 deg; joints [-7.166, -48.397, 79.945, -0.331, 60.611, 35.885, -22.883]
  MoveL 886 to (-42.45, 103.34, -101.62) mm, rotated rx -48.64 ry 0 rz -157.91 deg; joints [-7.179, -48.352, 79.975, -0.34, 60.611, 35.878, -22.959]
  MoveL 887 to (-41.64, 103.55, -101.74) mm, rotated rx -48.58 ry 0 rz -158.34 deg; joints [-7.19, -48.363, 79.998, -0.342, 60.612, 35.93, -22.548]
  MoveL 888 to (-40.85, 103.85, -101.76) mm, rotated rx -48.58 ry 0 rz -158.34 deg; joints [-7.19, -48.318, 80.003, -0.348, 60.612, 35.933, -22.598]
  MoveL 889 to (-39.94, 104.31, -101.64) mm, rotated rx -48.64 ry 0 rz -158.86 deg; joints [-7.179, -48.307, 79.982, -0.346, 60.612, 35.885, -22.065]
  MoveL 890 to (-39.97, 104.32, -101.62) mm, rotated rx -47.2 ry 0 rz -160.12 deg; joints [-7.348, -48.601, 80.305, -0.357, 60.612, 37.156, -20.832]
  MoveL 891 to (-40.46, 103.11, -102.66) mm, rotated rx -46.67 ry 0 rz -159.67 deg; joints [-7.447, -48.699, 80.507, -0.374, 60.613, 37.597, -21.386]
  MoveL 892 to (-40.5, 102.15, -103.6) mm, rotated rx -46.67 ry 0 rz -159.67 deg; joints [-7.481, -48.753, 80.575, -0.378, 60.613, 37.564, -21.401]
  MoveL 893 to (-40.38, 101.81, -103.97) mm, rotated rx -46.47 ry 0 rz -159.67 deg; joints [-7.518, -48.789, 80.651, -0.384, 60.613, 37.728, -21.443]
  MoveL 894 to (-39.8, 101.13, -104.86) mm, rotated rx -46.47 ry 0 rz -159.67 deg; joints [-7.55, -48.805, 80.719, -0.392, 60.613, 37.7, -21.496]
  MoveL 895 to (-37.19, 99.47, -107.37) mm, rotated rx -45.13 ry 0 rz -160.69 deg; joints [-7.796, -49.061, 81.241, -0.438, 60.613, 38.826, -20.748]
  MoveL 896 to (-36.15, 99.14, -108.04) mm, rotated rx -45.13 ry 0 rz -160.69 deg; joints [-7.819, -49.041, 81.298, -0.45, 60.613, 38.809, -20.826]
  MoveL 897 to (-35.88, 99.12, -108.15) mm, rotated rx -45.07 ry 0 rz -160.82 deg; joints [-7.83, -49.053, 81.322, -0.452, 60.613, 38.859, -20.704]
  MoveL 898 to (-35.2, 99.14, -108.35) mm, rotated rx -45.07 ry 0 rz -160.82 deg; joints [-7.837, -49.026, 81.341, -0.458, 60.613, 38.856, -20.751]
  MoveL 899 to (-31.81, 99.55, -109.02) mm, rotated rx -44.7 ry 0 rz -162.65 deg; joints [-7.903, -49.097, 81.486, -0.471, 60.613, 39.162, -18.994]
  MoveL 900 to (-31.5, 99.6, -109.07) mm, rotated rx -44.7 ry 0 rz -162.65 deg; joints [-7.905, -49.082, 81.491, -0.474, 60.613, 39.162, -19.014]
  MoveL 901 to (-31.19, 99.66, -109.1) mm, rotated rx -44.68 ry 0 rz -162.83 deg; joints [-7.908, -49.086, 81.498, -0.475, 60.614, 39.177, -18.846]
  MoveL 902 to (-29.78, 99.83, -109.33) mm, rotated rx -44.54 ry 0 rz -163.7 deg; joints [-7.933, -49.123, 81.551, -0.478, 60.614, 39.296, -17.991]
  MoveL 903 to (-29.79, 99.83, -109.32) mm, rotated rx -43.61 ry 0 rz -164.76 deg; joints [-8.039, -49.342, 81.774, -0.485, 60.614, 40.128, -16.934]
  MoveL 904 to (-29.36, 98.21, -110.91) mm, rotated rx -42.73 ry 0 rz -164.75 deg; joints [-8.196, -49.518, 82.125, -0.519, 60.614, 40.865, -17.118]
  MoveL 905 to (-29.24, 97.91, -111.2) mm, rotated rx -42.73 ry 0 rz -164.75 deg; joints [-8.206, -49.529, 82.15, -0.521, 60.614, 40.856, -17.133]
  MoveL 906 to (-28.73, 97.35, -111.82) mm, rotated rx -42.73 ry 0 rz -164.75 deg; joints [-8.229, -49.537, 82.206, -0.529, 60.614, 40.837, -17.18]
  MoveL 907 to (-28.33, 97.08, -112.16) mm, rotated rx -42.54 ry 0 rz -164.93 deg; joints [-8.263, -49.576, 82.282, -0.536, 60.614, 40.997, -17.043]
  MoveL 908 to (-31.85, 110.14, -126.89) mm, rotated rx -42.54 ry 0 rz -164.93 deg; joints [-8.723, -48.908, 80.918, -0.467, 60.614, 40.498, -16.346]
  Set speed (1000.0 mm/s)
  MoveL 909 to (-30.55, 107.92, -129.11) mm, rotated rx -41.19 ry 0 rz -165.43 deg; joints [-8.955, -49.192, 81.459, -0.518, 60.614, 41.648, -16.105]
  Set speed (5.0 mm/s)
  MoveL 910 to (-27.24, 95.17, -114.05) mm, rotated rx -41.19 ry 0 rz -165.43 deg; joints [-8.483, -49.853, 82.794, -0.584, 60.614, 42.157, -16.779]
  Set speed (16.7 mm/s)
  MoveL 911 to (-27.07, 94.92, -114.3) mm, rotated rx -41.04 ry 0 rz -165.49 deg; joints [-8.508, -49.884, 82.855, -0.59, 60.614, 42.281, -16.752]
  MoveL 912 to (-26.62, 94.47, -114.78) mm, rotated rx -41.04 ry 0 rz -165.49 deg; joints [-8.526, -49.889, 82.9, -0.597, 60.614, 42.267, -16.792]
  MoveL 913 to (-25.14, 93.4, -115.97) mm, rotated rx -40.33 ry 0 rz -166.19 deg; joints [-8.648, -50.042, 83.194, -0.626, 60.615, 42.87, -16.239]
  MoveL 914 to (-25.15, 93.43, -115.95) mm, rotated rx -39.74 ry 0 rz -166.41 deg; joints [-8.711, -50.14, 83.344, -0.638, 60.615, 43.405, -16.07]
  MoveL 915 to (-25.01, 92.14, -117.01) mm, rotated rx -39.11 ry 0 rz -166.31 deg; joints [-8.819, -50.278, 83.609, -0.665, 60.615, 43.942, -16.296]
  MoveL 916 to (-24.75, 91.45, -117.61) mm, rotated rx -39.11 ry 0 rz -166.31 deg; joints [-8.841, -50.304, 83.667, -0.672, 60.615, 43.923, -16.328]
  MoveL 917 to (-24.52, 91.12, -117.91) mm, rotated rx -38.93 ry 0 rz -166.4 deg; joints [-8.873, -50.345, 83.745, -0.68, 60.615, 44.081, -16.281]
  MoveL 918 to (-24, 90.62, -118.4) mm, rotated rx -38.93 ry 0 rz -166.4 deg; joints [-8.891, -50.349, 83.795, -0.688, 60.615, 44.067, -16.327]
  MoveL 919 to (-22.5, 89.61, -119.46) mm, rotated rx -38.27 ry 0 rz -167.16 deg; joints [-9.001, -50.497, 84.074, -0.717, 60.615, 44.629, -15.692]
  MoveL 920 to (-22.5, 89.65, -119.43) mm, rotated rx -37.03 ry 0 rz -166.95 deg; joints [-9.129, -50.653, 84.407, -0.755, 60.615, 45.765, -16.089]
  MoveL 921 to (-24.87, 86.81, -121.05) mm, rotated rx -36.02 ry 0 rz -165.09 deg; joints [-9.295, -50.889, 84.844, -0.801, 60.615, 46.63, -18.149]
  MoveL 922 to (-25.28, 85.96, -121.57) mm, rotated rx -36.02 ry 0 rz -165.09 deg; joints [-9.316, -50.946, 84.89, -0.803, 60.626, 46.61, -18.149]
  MoveL 923 to (-25.23, 85.07, -122.2) mm, rotated rx -36.02 ry 0 rz -165.09 deg; joints [-9.341, -50.991, 84.956, -0.809, 60.626, 46.588, -18.169]
  MoveL 924 to (-25.12, 84.72, -122.47) mm, rotated rx -35.85 ry 0 rz -165.11 deg; joints [-9.37, -51.033, 85.033, -0.817, 60.626, 46.739, -18.191]
  MoveL 925 to (-24.62, 83.97, -123.09) mm, rotated rx -35.85 ry 0 rz -165.11 deg; joints [-9.394, -51.053, 85.101, -0.827, 60.626, 46.72, -18.239]
  MoveL 926 to (-22.9, 82.39, -124.47) mm, rotated rx -34.92 ry 0 rz -165.95 deg; joints [-9.543, -51.276, 85.509, -0.871, 60.626, 47.525, -17.586]
  MoveL 927 to (-22.92, 82.41, -124.46) mm, rotated rx -34.46 ry 0 rz -166.13 deg; joints [-9.588, -51.358, 85.631, -0.882, 60.626, 47.942, -17.446]
  MoveL 928 to (-22.74, 81.54, -125.06) mm, rotated rx -34.05 ry 0 rz -166.11 deg; joints [-9.653, -51.458, 85.813, -0.901, 60.626, 48.296, -17.553]
  MoveL 929 to (-22.54, 81.02, -125.44) mm, rotated rx -34.05 ry 0 rz -166.11 deg; joints [-9.668, -51.478, 85.856, -0.907, 60.626, 48.284, -17.577]
  MoveL 930 to (-22.42, 80.81, -125.59) mm, rotated rx -33.95 ry 0 rz -166.15 deg; joints [-9.685, -51.504, 85.903, -0.912, 60.626, 48.376, -17.552]
  MoveL 931 to (-22.2, 80.51, -125.83) mm, rotated rx -33.95 ry 0 rz -166.15 deg; joints [-9.694, -51.511, 85.931, -0.916, 60.626, 48.369, -17.573]
  MoveL 932 to (-21.5, 79.72, -126.44) mm, rotated rx -33.51 ry 0 rz -166.49 deg; joints [-9.762, -51.618, 86.124, -0.938, 60.626, 48.746, -17.32]
  MoveL 933 to (-21.49, 79.74, -126.44) mm, rotated rx -32.68 ry 0 rz -166.42 deg; joints [-9.843, -51.742, 86.359, -0.964, 60.626, 49.518, -17.502]
  MoveL 934 to (-22.41, 77.11, -127.9) mm, rotated rx -31.66 ry 0 rz -165.36 deg; joints [-10.001, -52.003, 86.822, -1.016, 60.626, 50.408, -18.768]
  MoveL 935 to (-22.43, 77.01, -127.96) mm, rotated rx -31.53 ry 0 rz -165.22 deg; joints [-10.015, -52.02, 86.867, -1.022, 60.626, 50.526, -18.94]
  MoveL 936 to (-23.67, 74.16, -129.41) mm, rotated rx -30.49 ry 0 rz -163.81 deg; joints [-10.173, -52.292, 87.345, -1.076, 60.626, 51.44, -20.557]
  MoveL 937 to (-23.69, 74.17, -129.4) mm, rotated rx -30.27 ry 0 rz -163.37 deg; joints [-10.193, -52.297, 87.411, -1.088, 60.626, 51.647, -21.063]
  MoveL 938 to (-26.22, 70.97, -130.7) mm, rotated rx -29.31 ry 0 rz -160.89 deg; joints [-10.336, -52.555, 87.855, -1.138, 60.626, 52.486, -23.734]
  MoveL 939 to (-29.43, 80.22, -148.14) mm, rotated rx -29.31 ry 0 rz -160.89 deg; joints [-10.903, -51.968, 86.788, -1.117, 60.626, 51.903, -23.259]
  Set speed (1000.0 mm/s)
  MoveL 940 to (-28.39, 76.79, -150.15) mm, rotated rx -29.19 ry 0 rz -160.94 deg; joints [-11.001, -52.155, 87.097, -1.151, 60.626, 51.949, -23.333]
  Set speed (5.0 mm/s)
  MoveL 941 to (-25.2, 67.57, -132.69) mm, rotated rx -29.19 ry 0 rz -160.94 deg; joints [-10.433, -52.743, 88.159, -1.171, 60.627, 52.533, -23.803]
  Set speed (16.7 mm/s)
  MoveL 942 to (-23.44, 66.82, -133.39) mm, rotated rx -28.62 ry 0 rz -162.11 deg; joints [-10.514, -52.897, 88.422, -1.2, 60.627, 53.034, -22.742]
  MoveL 943 to (-22.89, 66.66, -133.57) mm, rotated rx -28.62 ry 0 rz -162.11 deg; joints [-10.522, -52.888, 88.452, -1.208, 60.627, 53.032, -22.781]
  MoveL 944 to (-21.54, 66.75, -133.74) mm, rotated rx -28.62 ry 0 rz -162.11 deg; joints [-10.528, -52.838, 88.49, -1.225, 60.627, 53.035, -22.871]
  MoveL 945 to (-21.39, 66.8, -133.74) mm, rotated rx -28.62 ry 0 rz -162.25 deg; joints [-10.528, -52.838, 88.49, -1.225, 60.627, 53.035, -22.735]
  MoveL 946 to (-21.09, 66.94, -133.72) mm, rotated rx -28.64 ry 0 rz -162.61 deg; joints [-10.526, -52.839, 88.481, -1.223, 60.627, 53.02, -22.358]
  MoveL 947 to (-20.32, 67.13, -133.74) mm, rotated rx -28.62 ry 0 rz -163.26 deg; joints [-10.528, -52.844, 88.488, -1.224, 60.627, 53.034, -21.717]
  MoveL 948 to (-19.09, 67.49, -133.74) mm, rotated rx -28.62 ry 0 rz -164.2 deg; joints [-10.528, -52.837, 88.49, -1.225, 60.626, 53.035, -20.779]
  MoveL 949 to (-18.33, 67.84, -133.67) mm, rotated rx -28.67 ry 0 rz -164.34 deg; joints [-10.52, -52.791, 88.473, -1.229, 60.626, 52.998, -20.669]
  MoveL 950 to (-17.72, 68.39, -133.48) mm, rotated rx -28.72 ry 0 rz -164.48 deg; joints [-10.506, -52.739, 88.437, -1.23, 60.626, 52.965, -20.545]
  MoveL 951 to (-14.72, 70.88, -132.54) mm, rotated rx -29.47 ry 0 rz -167.32 deg; joints [-10.397, -52.535, 88.084, -1.19, 60.626, 52.296, -17.555]
  MoveL 952 to (-14.46, 71.1, -132.45) mm, rotated rx -29.51 ry 0 rz -167.44 deg; joints [-10.389, -52.514, 88.063, -1.189, 60.626, 52.265, -17.432]
  MoveL 953 to (-14.22, 71.35, -132.34) mm, rotated rx -29.51 ry 0 rz -167.44 deg; joints [-10.385, -52.496, 88.055, -1.188, 60.616, 52.269, -17.434]
  MoveL 954 to (-13.06, 72.66, -131.75) mm, rotated rx -29.98 ry 0 rz -168.56 deg; joints [-10.316, -52.371, 87.837, -1.163, 60.616, 51.853, -16.224]
  MoveL 955 to (-12.27, 73.21, -131.52) mm, rotated rx -30.27 ry 0 rz -169.56 deg; joints [-10.279, -52.325, 87.718, -1.146, 60.616, 51.59, -15.147]
  MoveL 956 to (-11.79, 73.66, -131.31) mm, rotated rx -30.27 ry 0 rz -169.56 deg; joints [-10.27, -52.289, 87.704, -1.146, 60.6, 51.599, -15.152]
  MoveL 957 to (-11.6, 73.89, -131.2) mm, rotated rx -30.36 ry 0 rz -169.74 deg; joints [-10.257, -52.266, 87.663, -1.141, 60.6, 51.522, -14.957]
  MoveL 958 to (-11.34, 74.28, -131) mm, rotated rx -30.36 ry 0 rz -169.74 deg; joints [-10.249, -52.237, 87.642, -1.141, 60.597, 51.531, -14.962]
  MoveL 959 to (-9.75, 77.15, -129.46) mm, rotated rx -31.52 ry 0 rz -171.29 deg; joints [-10.074, -51.933, 87.107, -1.08, 60.597, 50.505, -13.176]
  MoveL 960 to (-8.68, 78.06, -128.99) mm, rotated rx -32.08 ry 0 rz -172.54 deg; joints [-10.002, -51.835, 86.883, -1.05, 60.597, 50.001, -11.797]
  MoveL 961 to (-8.12, 78.78, -128.59) mm, rotated rx -32.08 ry 0 rz -172.54 deg; joints [-9.985, -51.78, 86.845, -1.049, 60.586, 50.018, -11.804]
  MoveL 962 to (-8.05, 78.92, -128.51) mm, rotated rx -32.14 ry 0 rz -172.6 deg; joints [-9.976, -51.764, 86.817, -1.046, 60.586, 49.965, -11.727]
  MoveL 963 to (-7.91, 79.29, -128.29) mm, rotated rx -32.14 ry 0 rz -172.6 deg; joints [-9.966, -51.74, 86.792, -1.045, 60.586, 49.974, -11.727]
  MoveL 964 to (-7.49, 80.82, -127.35) mm, rotated rx -32.81 ry 0 rz -173.04 deg; joints [-9.863, -51.57, 86.489, -1.011, 60.586, 49.388, -11.155]
  MoveL 965 to (-6.64, 82.04, -126.62) mm, rotated rx -33.57 ry 0 rz -173.96 deg; joints [-9.759, -51.419, 86.184, -0.974, 60.586, 48.711, -10.071]
  MoveL 966 to (-6.48, 82.31, -126.45) mm, rotated rx -33.57 ry 0 rz -173.96 deg; joints [-9.753, -51.4, 86.167, -0.973, 60.584, 48.718, -10.071]
  MoveL 967 to (-6.28, 82.72, -126.19) mm, rotated rx -33.75 ry 0 rz -174.14 deg; joints [-9.724, -51.355, 86.086, -0.964, 60.584, 48.559, -9.861]
  MoveL 968 to (-6.17, 82.97, -126.04) mm, rotated rx -33.75 ry 0 rz -174.14 deg; joints [-9.718, -51.339, 86.069, -0.963, 60.584, 48.565, -9.86]
  MoveL 969 to (-4.86, 86.58, -123.64) mm, rotated rx -35.38 ry 0 rz -175.25 deg; joints [-9.459, -50.942, 85.345, -0.883, 60.584, 47.15, -8.415]
  MoveL 970 to (-4.77, 87.47, -123.02) mm, rotated rx -35.38 ry 0 rz -175.25 deg; joints [-9.434, -50.897, 85.279, -0.877, 60.584, 47.172, -8.393]
  MoveL 971 to (-4.81, 87.73, -122.83) mm, rotated rx -35.51 ry 0 rz -175.23 deg; joints [-9.414, -50.867, 85.224, -0.871, 60.584, 47.064, -8.381]
  MoveL 972 to (-4.87, 87.98, -122.65) mm, rotated rx -35.51 ry 0 rz -175.23 deg; joints [-9.407, -50.859, 85.204, -0.869, 60.584, 47.07, -8.369]
  MoveL 973 to (-5.21, 89.02, -121.87) mm, rotated rx -36 ry 0 rz -175.07 deg; joints [-9.326, -50.741, 84.986, -0.845, 60.583, 46.642, -8.43]
  MoveL 974 to (-5.24, 89.01, -121.88) mm, rotated rx -36.91 ry 0 rz -175.6 deg; joints [-9.234, -50.651, 84.732, -0.81, 60.583, 45.807, -7.738]
  MoveL 975 to (-4.26, 89.78, -121.36) mm, rotated rx -37.25 ry 0 rz -176.26 deg; joints [-9.179, -50.573, 84.585, -0.794, 60.583, 45.517, -7.001]
  MoveL 976 to (-3.87, 90.15, -121.1) mm, rotated rx -37.25 ry 0 rz -176.26 deg; joints [-9.169, -50.544, 84.567, -0.794, 60.572, 45.527, -7.001]
  MoveL 977 to (-3.46, 91.17, -120.34) mm, rotated rx -37.25 ry 0 rz -176.26 deg; joints [-9.138, -50.478, 84.493, -0.79, 60.572, 45.555, -6.993]
  MoveL 978 to (-3.45, 91.36, -120.21) mm, rotated rx -37.33 ry 0 rz -176.28 deg; joints [-9.124, -50.458, 84.456, -0.786, 60.572, 45.48, -6.961]
  MoveL 979 to (-3.51, 91.87, -119.81) mm, rotated rx -37.33 ry 0 rz -176.28 deg; joints [-9.109, -50.437, 84.415, -0.781, 60.572, 45.493, -6.94]
  MoveL 980 to (-4.01, 93.64, -118.41) mm, rotated rx -38.19 ry 0 rz -176.04 deg; joints [-8.965, -50.242, 84.046, -0.742, 60.572, 44.757, -6.999]
  MoveL 981 to (-4, 93.62, -118.43) mm, rotated rx -38.58 ry 0 rz -176.07 deg; joints [-8.926, -50.191, 83.945, -0.731, 60.572, 44.407, -6.919]
  MoveL 982 to (-3.66, 94.95, -117.38) mm, rotated rx -39.22 ry 0 rz -176.33 deg; joints [-8.817, -50.048, 83.672, -0.702, 60.572, 43.858, -6.525]
  MoveL 983 to (-4.47, 107.57, -132.88) mm, rotated rx -39.22 ry 0 rz -176.33 deg; joints [-9.305, -49.394, 82.376, -0.644, 60.572, 43.336, -5.883]
  Set speed (1000.0 mm/s)
  MoveL 984 to (-3.83, 110.44, -130.52) mm, rotated rx -40.44 ry 0 rz -176.75 deg; joints [-9.085, -49.119, 81.832, -0.587, 60.572, 42.306, -5.19]
  Set speed (5.0 mm/s)
  MoveL 985 to (-3.09, 97.49, -115.3) mm, rotated rx -40.44 ry 0 rz -176.75 deg; joints [-8.607, -49.779, 83.155, -0.649, 60.571, 42.819, -5.853]
  Set speed (16.7 mm/s)
  MoveL 986 to (-2.24, 100.79, -112.45) mm, rotated rx -42.09 ry 0 rz -177.35 deg; joints [-8.32, -49.429, 82.471, -0.58, 60.571, 41.415, -4.919]
  MoveL 987 to (-2.17, 101.07, -112.19) mm, rotated rx -42.21 ry 0 rz -177.39 deg; joints [-8.297, -49.401, 82.418, -0.575, 60.571, 41.312, -4.854]
  MoveL 988 to (-1.61, 103.2, -110.24) mm, rotated rx -43.32 ry 0 rz -177.75 deg; joints [-8.102, -49.177, 81.972, -0.532, 60.571, 40.381, -4.264]
  MoveL 989 to (-1.56, 103.61, -109.86) mm, rotated rx -43.32 ry 0 rz -177.75 deg; joints [-8.088, -49.157, 81.94, -0.529, 60.571, 40.394, -4.251]
  MoveL 990 to (-1.57, 103.74, -109.74) mm, rotated rx -43.39 ry 0 rz -177.75 deg; joints [-8.075, -49.143, 81.912, -0.526, 60.571, 40.334, -4.237]
  MoveL 991 to (-1.73, 104.85, -108.68) mm, rotated rx -44.18 ry 0 rz -177.72 deg; joints [-7.948, -49.004, 81.627, -0.499, 60.571, 39.659, -4.119]
  MoveL 992 to (0.21, 108.08, -105.48) mm, rotated rx -46.08 ry 0 rz -178.91 deg; joints [-7.614, -48.657, 80.904, -0.431, 60.571, 38.047, -2.555]
  MoveL 993 to (0.42, 108.82, -104.72) mm, rotated rx -46.08 ry 0 rz -178.91 deg; joints [-7.586, -48.617, 80.846, -0.428, 60.571, 38.073, -2.538]
  MoveL 994 to (0.42, 109, -104.52) mm, rotated rx -46.19 ry 0 rz -178.9 deg; joints [-7.567, -48.598, 80.807, -0.424, 60.571, 37.987, -2.519]
  MoveL 995 to (0.32, 109.44, -104.07) mm, rotated rx -46.19 ry 0 rz -178.9 deg; joints [-7.55, -48.585, 80.772, -0.42, 60.571, 38.002, -2.496]
  MoveL 996 to (-0.31, 110.94, -102.46) mm, rotated rx -47.02 ry 0 rz -178.59 deg; joints [-7.396, -48.431, 80.452, -0.392, 60.571, 37.308, -2.638]
  MoveL 997 to (-0.3, 112.04, -101.27) mm, rotated rx -47.89 ry 0 rz -178.57 deg; joints [-7.251, -48.285, 80.159, -0.368, 60.571, 36.566, -2.518]
  MoveL 998 to (-0.34, 112.34, -100.94) mm, rotated rx -47.89 ry 0 rz -178.57 deg; joints [-7.239, -48.275, 80.135, -0.365, 60.571, 36.576, -2.503]
  MoveL 999 to (-0.39, 112.51, -100.74) mm, rotated rx -48 ry 0 rz -178.54 deg; joints [-7.22, -48.257, 80.097, -0.362, 60.57, 36.493, -2.506]
  MoveL 1000 to (-0.45, 112.67, -100.56) mm, rotated rx -48 ry 0 rz -178.54 deg; joints [-7.214, -48.254, 80.084, -0.361, 60.57, 36.498, -2.495]
  MoveL 1001 to (-1.06, 113.99, -99.05) mm, rotated rx -49.06 ry 0 rz -178.21 deg; joints [-7.035, -48.081, 79.73, -0.332, 60.57, 35.594, -2.645]
  MoveL 1002 to (-0.89, 116.98, -95.51) mm, rotated rx -51.11 ry 0 rz -178.43 deg; joints [-6.664, -47.76, 79.026, -0.276, 60.57, 33.886, -2.044]
  MoveL 1003 to (0.74, 119.64, -92.16) mm, rotated rx -52.74 ry 0 rz -179.24 deg; joints [-6.35, -47.497, 78.455, -0.234, 60.569, 32.553, -0.915]
  MoveL 1004 to (0.91, 120.12, -91.53) mm, rotated rx -52.74 ry 0 rz -179.24 deg; joints [-6.327, -47.469, 78.416, -0.232, 60.569, 32.574, -0.904]
  MoveL 1005 to (0.92, 120.24, -91.37) mm, rotated rx -52.82 ry 0 rz -179.25 deg; joints [-6.312, -47.457, 78.39, -0.231, 60.569, 32.511, -0.884]
  MoveL 1006 to (0.92, 120.42, -91.13) mm, rotated rx -52.82 ry 0 rz -179.25 deg; joints [-6.304, -47.45, 78.375, -0.23, 60.569, 32.519, -0.876]
  MoveL 1007 to (0.75, 121.59, -89.57) mm, rotated rx -53.74 ry 0 rz -179.18 deg; joints [-6.135, -47.318, 78.082, -0.21, 60.569, 31.748, -0.779]
  MoveL 1008 to (1.24, 122.75, -87.97) mm, rotated rx -54.6 ry 0 rz -179.45 deg; joints [-5.974, -47.197, 77.807, -0.192, 60.569, 31.041, -0.362]
  MoveL 1009 to (1.31, 123.04, -87.57) mm, rotated rx -54.6 ry 0 rz -179.45 deg; joints [-5.96, -47.182, 77.784, -0.19, 60.569, 31.054, -0.354]
  MoveL 1010 to (1.32, 123.17, -87.37) mm, rotated rx -54.69 ry 0 rz -179.45 deg; joints [-5.942, -47.169, 77.754, -0.189, 60.569, 30.981, -0.331]
  MoveL 1011 to (1.3, 123.44, -87) mm, rotated rx -54.69 ry 0 rz -179.45 deg; joints [-5.929, -47.16, 77.732, -0.187, 60.568, 30.993, -0.318]
  MoveL 1012 to (1, 124.63, -85.29) mm, rotated rx -55.56 ry 0 rz -179.31 deg; joints [-5.762, -47.035, 77.456, -0.17, 60.568, 30.284, -0.307]
  MoveL 1013 to (0.97, 124.77, -85.09) mm, rotated rx -55.76 ry 0 rz -179.3 deg; joints [-5.73, -47.012, 77.404, -0.167, 60.568, 30.112, -0.29]
  MoveL 1014 to (1.26, 127.48, -80.96) mm, rotated rx -57.64 ry 0 rz -179.45 deg; joints [-5.352, -46.749, 76.808, -0.134, 60.568, 28.598, 0.192]
  MoveL 1015 to (1.26, 127.68, -80.64) mm, rotated rx -57.64 ry 0 rz -179.45 deg; joints [-5.341, -46.742, 76.791, -0.133, 60.568, 28.608, 0.202]
  MoveL 1016 to (1.24, 127.76, -80.51) mm, rotated rx -57.7 ry 0 rz -179.44 deg; joints [-5.329, -46.734, 76.774, -0.133, 60.568, 28.562, 0.206]
  MoveL 1017 to (1.19, 127.95, -80.22) mm, rotated rx -57.7 ry 0 rz -179.44 deg; joints [-5.32, -46.73, 76.758, -0.131, 60.567, 28.572, 0.218]
  MoveL 1018 to (0.96, 128.4, -79.5) mm, rotated rx -58.28 ry 0 rz -179.32 deg; joints [-5.222, -46.685, 76.632, -0.121, 60.526, 28.085, 0.218]
  MoveL 1019 to (0.97, 128.48, -79.36) mm, rotated rx -58.34 ry 0 rz -179.32 deg; joints [-5.21, -46.678, 76.613, -0.12, 60.525, 28.037, 0.232]
  MoveL 1020 to (1.52, 130.36, -76.23) mm, rotated rx -59.82 ry 0 rz -179.58 deg; joints [-4.913, -46.49, 76.178, -0.101, 60.525, 26.837, 0.745]
  MoveL 1021 to (1.55, 130.51, -75.97) mm, rotated rx -59.82 ry 0 rz -179.58 deg; joints [-4.904, -46.484, 76.165, -0.1, 60.524, 26.846, 0.752]
  MoveL 1022 to (1.57, 130.9, -75.29) mm, rotated rx -60.12 ry 0 rz -179.59 deg; joints [-4.843, -46.446, 76.078, -0.097, 60.524, 26.61, 0.81]
  MoveL 1023 to (1.66, 133.76, -70.09) mm, rotated rx -62.52 ry 0 rz -179.66 deg; joints [-4.355, -46.164, 75.411, -0.073, 60.524, 24.679, 1.264]
  MoveL 1024 to (1.75, 133.98, -69.66) mm, rotated rx -62.71 ry 0 rz -179.7 deg; joints [-4.317, -46.143, 75.361, -0.072, 60.524, 24.534, 1.332]
  MoveL 1025 to (2.41, 135.04, -67.57) mm, rotated rx -63.67 ry 0 rz 180 deg; joints [-4.12, -46.04, 75.107, -0.065, 60.524, 23.76, 1.785]
  MoveL 1026 to (3, 135.96, -65.67) mm, rotated rx -64.48 ry 0 rz 179.75 deg; joints [-3.95, -45.951, 74.896, -0.06, 60.524, 23.122, 2.16]
  MoveL 1027 to (2.98, 135.95, -65.68) mm, rotated rx -65 ry 0 rz 179.34 deg; joints [-3.882, -45.971, 74.813, -0.056, 60.524, 22.67, 2.668]
  MoveL 1028 to (7.92, 137.22, -62.57) mm, rotated rx -66.39 ry 0 rz 177.12 deg; joints [-3.593, -45.854, 74.47, -0.05, 60.524, 21.561, 5.123]
  MoveL 1029 to (8.14, 137.25, -62.48) mm, rotated rx -66.43 ry 0 rz 177.02 deg; joints [-3.585, -45.85, 74.461, -0.05, 60.524, 21.532, 5.22]
  MoveL 1030 to (11.32, 137.44, -61.55) mm, rotated rx -66.85 ry 0 rz 175.61 deg; joints [-3.498, -45.822, 74.361, -0.049, 60.523, 21.198, 6.705]
  MoveL 1031 to (11.54, 137.46, -61.48) mm, rotated rx -66.85 ry 0 rz 175.61 deg; joints [-3.495, -45.812, 74.361, -0.049, 60.518, 21.201, 6.7]
  MoveL 1032 to (12.41, 137.53, -61.14) mm, rotated rx -66.99 ry 0 rz 175.25 deg; joints [-3.465, -45.798, 74.327, -0.049, 60.518, 21.09, 7.08]
  MoveL 1033 to (12.81, 137.58, -60.95) mm, rotated rx -66.99 ry 0 rz 175.25 deg; joints [-3.459, -45.781, 74.327, -0.049, 60.504, 21.096, 7.076]
  MoveL 1034 to (16.95, 138.2, -58.48) mm, rotated rx -68.01 ry 0 rz 173.57 deg; joints [-3.24, -45.684, 74.087, -0.048, 60.503, 20.294, 8.903]
  MoveL 1035 to (21.14, 138.65, -56) mm, rotated rx -69.03 ry 0 rz 171.89 deg; joints [-3.02, -45.603, 73.866, -0.048, 60.478, 19.494, 10.751]
  MoveL 1036 to (22.1, 138.9, -55.01) mm, rotated rx -69.03 ry 0 rz 171.89 deg; joints [-2.987, -45.575, 73.866, -0.048, 60.416, 19.526, 10.785]
  MoveL 1037 to (22.2, 138.96, -54.82) mm, rotated rx -69.11 ry 0 rz 171.85 deg; joints [-2.97, -45.572, 73.853, -0.048, 60.409, 19.466, 10.84]
  MoveL 1038 to (22.35, 139.07, -54.48) mm, rotated rx -69.11 ry 0 rz 171.85 deg; joints [-2.959, -45.571, 73.852, -0.048, 60.39, 19.477, 10.859]
  MoveL 1039 to (22.88, 139.59, -52.91) mm, rotated rx -69.96 ry 0 rz 171.57 deg; joints [-2.793, -45.571, 73.734, -0.047, 60.298, 18.794, 11.346]
  MoveL 1040 to (25.99, 140.24, -49.64) mm, rotated rx -71.43 ry 0 rz 170.26 deg; joints [-2.485, -45.57, 73.535, -0.049, 60.125, 17.631, 13.029]
  MoveL 1041 to (26.74, 140.41, -48.75) mm, rotated rx -71.74 ry 0 rz 170.01 deg; joints [-2.414, -45.57, 73.498, -0.05, 60.072, 17.394, 13.365]
  MoveL 1042 to (32.5, 141.63, -41.13) mm, rotated rx -74.73 ry 0 rz 167.89 deg; joints [-1.751, -45.57, 73.148, -0.074, 59.694, 15.076, 16.217]
  MoveL 1043 to (32.75, 141.66, -40.84) mm, rotated rx -74.89 ry 0 rz 167.76 deg; joints [-1.719, -45.57, 73.128, -0.076, 59.686, 14.948, 16.374]
  MoveL 1044 to (35.63, 141.87, -37.54) mm, rotated rx -76.2 ry 0 rz 166.66 deg; joints [-1.428, -45.57, 72.988, -0.092, 59.548, 13.933, 17.751]
  MoveL 1045 to (38.54, 141.6, -35.67) mm, rotated rx -77.13 ry 0 rz 165.32 deg; joints [-1.238, -45.57, 72.875, -0.105, 59.514, 13.208, 19.242]
  MoveL 1046 to (38.93, 141.57, -35.36) mm, rotated rx -77.13 ry 0 rz 165.32 deg; joints [-1.228, -45.554, 72.875, -0.106, 59.499, 13.218, 19.241]
  MoveL 1047 to (39.55, 141.62, -34.44) mm, rotated rx -77.13 ry 0 rz 165.32 deg; joints [-1.198, -45.537, 72.875, -0.108, 59.459, 13.249, 19.264]
  MoveL 1048 to (39.7, 141.67, -34.05) mm, rotated rx -77.28 ry 0 rz 165.26 deg; joints [-1.163, -45.536, 72.86, -0.11, 59.446, 13.132, 19.346]
  MoveL 1049 to (41.12, 142.09, -30.47) mm, rotated rx -78.67 ry 0 rz 164.78 deg; joints [-0.851, -45.535, 72.732, -0.134, 59.317, 12.065, 20.091]
  MoveL 1050 to (41.26, 142.16, -29.95) mm, rotated rx -78.67 ry 0 rz 164.78 deg; joints [-0.834, -45.535, 72.731, -0.136, 59.299, 12.083, 20.109]
  MoveL 1051 to (41.16, 142.43, -28.75) mm, rotated rx -78.67 ry 0 rz 164.78 deg; joints [-0.795, -45.536, 72.708, -0.139, 59.299, 12.124, 20.133]
  MoveL 1052 to (41.03, 142.55, -28.37) mm, rotated rx -78.82 ry 0 rz 164.84 deg; joints [-0.761, -45.536, 72.695, -0.142, 59.286, 12.009, 20.097]
  MoveL 1053 to (40.52, 142.86, -27.52) mm, rotated rx -78.82 ry 0 rz 164.84 deg; joints [-0.733, -45.563, 72.681, -0.144, 59.286, 12.038, 20.138]
  MoveL 1054 to (38.89, 143.61, -25.84) mm, rotated rx -79.47 ry 0 rz 165.52 deg; joints [-0.587, -45.563, 72.627, -0.157, 59.233, 11.543, 19.567]
  MoveL 1055 to (38.92, 143.6, -25.89) mm, rotated rx -80.77 ry 0 rz 165.54 deg; joints [-0.404, -45.563, 72.568, -0.174, 59.16, 10.426, 19.675]
  MoveL 1056 to (39.51, 143.55, -25.27) mm, rotated rx -81.01 ry 0 rz 165.32 deg; joints [-0.35, -45.563, 72.55, -0.179, 59.142, 10.245, 19.935]
  MoveL 1057 to (40.07, 143.56, -24.36) mm, rotated rx -81.01 ry 0 rz 165.32 deg; joints [-0.32, -45.545, 72.55, -0.182, 59.11, 10.277, 19.949]
  MoveL 1058 to (40.29, 143.6, -23.74) mm, rotated rx -81.25 ry 0 rz 165.24 deg; joints [-0.267, -45.544, 72.532, -0.187, 59.093, 10.098, 20.06]
  MoveL 1059 to (40.41, 143.65, -23.24) mm, rotated rx -81.25 ry 0 rz 165.24 deg; joints [-0.25, -45.544, 72.532, -0.189, 59.078, 10.115, 20.075]
  MoveL 1060 to (40.3, 143.86, -22.08) mm, rotated rx -81.25 ry 0 rz 165.24 deg; joints [-0.212, -45.546, 72.513, -0.192, 59.078, 10.155, 20.096]
  MoveL 1061 to (38.72, 144.91, -17.54) mm, rotated rx -82.98 ry 0 rz 165.93 deg; joints [0.183, -45.546, 72.397, -0.232, 58.961, 8.833, 19.644]
  MoveL 1062 to (38.58, 144.99, -17.22) mm, rotated rx -82.98 ry 0 rz 165.93 deg; joints [0.194, -45.553, 72.393, -0.234, 58.961, 8.844, 19.655]
  MoveL 1063 to (38.48, 145.04, -17.03) mm, rotated rx -83.05 ry 0 rz 165.97 deg; joints [0.21, -45.553, 72.389, -0.235, 58.957, 8.791, 19.623]
  MoveL 1064 to (37.63, 145.45, -15.32) mm, rotated rx -83.73 ry 0 rz 166.33 deg; joints [0.362, -45.553, 72.35, -0.252, 58.915, 8.276, 19.338]
  MoveL 1065 to (37.23, 145.61, -14.75) mm, rotated rx -83.73 ry 0 rz 166.33 deg; joints [0.38, -45.575, 72.345, -0.254, 58.915, 8.296, 19.365]
  MoveL 1066 to (37.03, 145.69, -14.54) mm, rotated rx -83.81 ry 0 rz 166.42 deg; joints [0.399, -45.575, 72.341, -0.256, 58.91, 8.234, 19.293]
  MoveL 1067 to (36.58, 145.84, -14.17) mm, rotated rx -83.81 ry 0 rz 166.42 deg; joints [0.412, -45.6, 72.339, -0.259, 58.91, 8.247, 19.321]
  MoveL 1068 to (34.46, 146.47, -12.81) mm, rotated rx -84.32 ry 0 rz 167.26 deg; joints [0.529, -45.6, 72.31, -0.271, 58.882, 7.856, 18.533]
  MoveL 1069 to (34.47, 146.47, -12.84) mm, rotated rx -84.6 ry 0 rz 167.55 deg; joints [0.568, -45.569, 72.31, -0.275, 58.849, 7.619, 18.243]
  MoveL 1070 to (33.46, 146.84, -11.22) mm, rotated rx -85.22 ry 0 rz 167.96 deg; joints [0.709, -45.569, 72.279, -0.291, 58.818, 7.151, 17.9]
  MoveL 1071 to (33.09, 146.96, -10.77) mm, rotated rx -85.22 ry 0 rz 167.96 deg; joints [0.724, -45.589, 72.276, -0.293, 58.818, 7.167, 17.923]
  MoveL 1072 to (32.68, 147.08, -10.37) mm, rotated rx -85.37 ry 0 rz 168.12 deg; joints [0.758, -45.589, 72.269, -0.297, 58.81, 7.052, 17.775]
  MoveL 1073 to (32.51, 147.13, -10.22) mm, rotated rx -85.37 ry 0 rz 168.12 deg; joints [0.764, -45.599, 72.268, -0.298, 58.81, 7.057, 17.786]
  MoveL 1074 to (29.75, 147.84, -8.03) mm, rotated rx -86.2 ry 0 rz 169.2 deg; joints [0.954, -45.599, 72.231, -0.319, 58.773, 6.427, 16.78]
  MoveL 1075 to (29.76, 147.84, -8.04) mm, rotated rx -86.94 ry 0 rz 169.57 deg; joints [1.059, -45.568, 72.231, -0.331, 58.71, 5.797, 16.448]
  MoveL 1076 to (29.76, 148.04, -2.01) mm, rotated rx -89.23 ry 0 rz 169.58 deg; joints [1.584, -45.568, 72.155, -0.391, 58.629, 4.063, 16.594]
  MoveL 1077 to (29.74, 148.04, -2.09) mm, rotated rx -89.77 ry 0 rz 169.41 deg; joints [1.659, -45.591, 72.144, -0.401, 58.629, 3.604, 16.802]
  MoveL 1078 to (31.21, 147.76, -0.05) mm, rotated rx -90.54 ry 0 rz 168.84 deg; joints [1.837, -45.591, 72.127, -0.421, 58.609, 3.018, 17.409]
  MoveL 1079 to (31.48, 147.7, 0.47) mm, rotated rx -90.85 ry 0 rz 168.64 deg; joints [1.898, -45.602, 72.12, -0.428, 58.609, 2.775, 17.626]
  MoveL 1080 to (32.83, 147.39, 1.86) mm, rotated rx -91.38 ry 0 rz 168.12 deg; joints [2.019, -45.602, 72.111, -0.442, 58.599, 2.377, 18.17]
  MoveL 1081 to (32.8, 147.39, 1.84) mm, rotated rx -91.48 ry 0 rz 166.92 deg; joints [2.036, -45.766, 72.111, -0.453, 58.635, 2.292, 19.497]
  MoveL 1082 to (33.53, 147.24, 1.33) mm, rotated rx -91.29 ry 0 rz 166.63 deg; joints [1.992, -45.766, 72.114, -0.448, 58.639, 2.439, 19.774]
  MoveL 1083 to (33.53, 147.25, 1.3) mm, rotated rx -91.01 ry 0 rz 166.38 deg; joints [1.952, -45.798, 72.114, -0.444, 58.655, 2.671, 20.043]
  MoveL 1084 to (34.87, 146.94, -0.79) mm, rotated rx -90.22 ry 0 rz 165.86 deg; joints [1.77, -45.798, 72.129, -0.423, 58.673, 3.27, 20.53]
  MoveL 1085 to (35.62, 146.75, -1.54) mm, rotated rx -90.22 ry 0 rz 165.86 deg; joints [1.744, -45.756, 72.129, -0.418, 58.67, 3.242, 20.491]
  MoveL 1086 to (36.61, 146.5, -1.89) mm, rotated rx -90.22 ry 0 rz 165.86 deg; joints [1.732, -45.702, 72.129, -0.414, 58.66, 3.228, 20.447]
  MoveL 1087 to (37.17, 146.36, -1.96) mm, rotated rx -90.2 ry 0 rz 165.64 deg; joints [1.726, -45.702, 72.13, -0.413, 58.661, 3.247, 20.663]
  MoveL 1088 to (37.6, 146.25, -1.97) mm, rotated rx -90.2 ry 0 rz 165.64 deg; joints [1.725, -45.68, 72.13, -0.412, 58.655, 3.246, 20.646]
  MoveL 1089 to (38.54, 146.01, -1.71) mm, rotated rx -90.2 ry 0 rz 165.64 deg; joints [1.733, -45.631, 72.13, -0.411, 58.641, 3.253, 20.611]
  MoveL 1090 to (42.69, 144.86, 0.45) mm, rotated rx -91.02 ry 0 rz 164.01 deg; joints [1.922, -45.631, 72.113, -0.432, 58.622, 2.631, 22.284]
  MoveL 1091 to (45.11, 144.13, 0.77) mm, rotated rx -91.23 ry 0 rz 162.75 deg; joints [1.964, -45.675, 72.113, -0.44, 58.622, 2.461, 23.589]
  MoveL 1092 to (59.93, 191.86, 1.85) mm, rotated rx -91.23 ry 0 rz 162.75 deg; joints [1.978, -45.675, 68.995, -0.863, 56.112, 2.674, 29.23]
  Set speed (5.0 mm/s)
  Call SetCLW
  Call SetRPM(70.0)
  MoveL 1093 to (-167.66, 48.48, 99.74) mm, rotated rx -119.08 ry 0 rz -105.84 deg; joints [9.059, -45.675, 71.189, -1.671, 57.352, -17.69, -65.497]
  MoveL 1094 to (-125.62, 36.55, 75.44) mm, rotated rx -119.08 ry 0 rz -105.84 deg; joints [8.418, -47.356, 75.594, -1.008, 57.352, -18.632, -68.284]
  Set speed (16.7 mm/s)
  MoveL 1095 to (-125.66, 36.09, 75.59) mm, rotated rx -119.15 ry 0 rz -105.64 deg; joints [8.432, -47.361, 75.608, -1.007, 57.352, -18.683, -68.494]
  MoveL 1096 to (-126.55, 30.63, 76.51) mm, rotated rx -119.51 ry 0 rz -103.41 deg; joints [8.514, -47.413, 75.689, -1.007, 57.359, -18.962, -70.763]
  MoveL 1097 to (-126.75, 29.66, 76.56) mm, rotated rx -119.51 ry 0 rz -103.13 deg; joints [8.518, -47.43, 75.689, -1.009, 57.368, -18.966, -71.03]
  MoveL 1098 to (-128.06, 23.4, 76.55) mm, rotated rx -119.51 ry 0 rz -100.36 deg; joints [8.516, -47.434, 75.687, -1.01, 57.368, -18.959, -73.798]
  MoveL 1099 to (-128.14, 21.08, 77.09) mm, rotated rx -119.77 ry 0 rz -99.07 deg; joints [8.57, -47.42, 75.74, -1.001, 57.369, -19.176, -75.151]
  MoveL 1100 to (-128.27, 20.02, 77.16) mm, rotated rx -119.78 ry 0 rz -98.84 deg; joints [8.574, -47.447, 75.74, -1.004, 57.38, -19.175, -75.364]
  MoveL 1101 to (-129.21, 15.23, 76.67) mm, rotated rx -119.57 ry 0 rz -96.86 deg; joints [8.529, -47.449, 75.696, -1.01, 57.38, -19.008, -77.305]
  MoveL 1102 to (-129.09, 12.94, 77.31) mm, rotated rx -119.88 ry 0 rz -95.42 deg; joints [8.591, -47.417, 75.756, -0.997, 57.38, -19.263, -78.839]
  MoveL 1103 to (-129.13, 12.06, 77.39) mm, rotated rx -119.88 ry 0 rz -95.42 deg; joints [8.595, -47.461, 75.756, -1.003, 57.395, -19.256, -78.809]
  MoveL 1104 to (-129.47, 10.56, 77.03) mm, rotated rx -119.87 ry 0 rz -95.25 deg; joints [8.584, -47.522, 75.749, -1.016, 57.395, -19.25, -78.905]
  MoveL 1105 to (-130.4, 8.24, 75.73) mm, rotated rx -119.29 ry 0 rz -94.2 deg; joints [8.461, -47.473, 75.622, -1.021, 57.395, -18.796, -79.881]
  MoveL 1106 to (-131.29, 7.17, 74.28) mm, rotated rx -119.29 ry 0 rz -94.2 deg; joints [8.412, -47.519, 75.579, -1.035, 57.395, -18.838, -79.791]
  MoveL 1107 to (-131.73, 7.15, 73.51) mm, rotated rx -119.24 ry 0 rz -94.19 deg; joints [8.379, -47.508, 75.546, -1.036, 57.395, -18.822, -79.78]
  MoveL 1108 to (-132.2, 7.3, 72.65) mm, rotated rx -118.87 ry 0 rz -94.24 deg; joints [8.298, -47.478, 75.466, -1.038, 57.395, -18.527, -79.681]
  MoveL 1109 to (-132.78, 6.62, 71.65) mm, rotated rx -117.86 ry 0 rz -93.79 deg; joints [8.126, -47.398, 75.299, -1.039, 57.395, -17.687, -80.042]
  MoveL 1110 to (-133.74, 6.48, 69.85) mm, rotated rx -117.86 ry 0 rz -93.79 deg; joints [8.064, -47.397, 75.252, -1.046, 57.377, -17.746, -79.977]
  MoveL 1111 to (-134.44, 7.5, 68.38) mm, rotated rx -116.1 ry 0 rz -93.73 deg; joints [7.774, -47.26, 75.007, -1.046, 57.335, -16.285, -79.887]
  MoveL 1112 to (-134.6, 7.01, 68.11) mm, rotated rx -115.99 ry 0 rz -93.52 deg; joints [7.749, -47.252, 74.985, -1.046, 57.335, -16.197, -80.086]
  MoveL 1113 to (-135.14, 4.27, 67.26) mm, rotated rx -115.55 ry 0 rz -92.15 deg; joints [7.659, -47.21, 74.918, -1.046, 57.312, -15.847, -81.404]
  MoveL 1114 to (-135.12, 2.4, 67.41) mm, rotated rx -115.57 ry 0 rz -90.95 deg; joints [7.664, -47.157, 74.918, -1.036, 57.31, -15.861, -82.666]
  MoveL 1115 to (-135.16, 1.48, 67.35) mm, rotated rx -115.54 ry 0 rz -90.76 deg; joints [7.66, -47.183, 74.917, -1.041, 57.31, -15.841, -82.823]
  MoveL 1116 to (-135.48, -0.78, 66.72) mm, rotated rx -115.35 ry 0 rz -90 deg; joints [7.613, -47.196, 74.879, -1.046, 57.31, -15.696, -83.534]
  MoveL 1117 to (-135.78, -3.03, 66.05) mm, rotated rx -115.03 ry 0 rz -89.05 deg; joints [7.546, -47.176, 74.824, -1.046, 57.308, -15.442, -84.446]
  MoveL 1118 to (-135.91, -3.72, 65.73) mm, rotated rx -115.03 ry 0 rz -89.05 deg; joints [7.537, -47.213, 74.82, -1.052, 57.308, -15.449, -84.405]
  MoveL 1119 to (-136.03, -4.12, 65.47) mm, rotated rx -114.92 ry 0 rz -88.88 deg; joints [7.512, -47.206, 74.801, -1.052, 57.307, -15.362, -84.562]
  MoveL 1120 to (-136.91, -6.5, 63.38) mm, rotated rx -114.14 ry 0 rz -88.02 deg; joints [7.334, -47.172, 74.66, -1.053, 57.306, -14.763, -85.318]
  MoveL 1121 to (-136.91, -6.56, 63.38) mm, rotated rx -113.87 ry 0 rz -87.34 deg; joints [7.295, -47.112, 74.66, -1.052, 57.234, -14.528, -85.983]
  MoveL 1122 to (-136.87, -8.62, 63.24) mm, rotated rx -113.81 ry 0 rz -86.48 deg; joints [7.282, -47.108, 74.649, -1.052, 57.232, -14.479, -86.837]
  MoveL 1123 to (-136.9, -9.7, 63.03) mm, rotated rx -113.75 ry 0 rz -86.19 deg; joints [7.267, -47.126, 74.64, -1.055, 57.232, -14.429, -87.099]
  MoveL 1124 to (-137.08, -13.18, 61.94) mm, rotated rx -113.32 ry 0 rz -84.85 deg; joints [7.171, -47.115, 74.571, -1.055, 57.231, -14.1, -88.382]
  MoveL 1125 to (-137.06, -13.23, 61.99) mm, rotated rx -113.99 ry 0 rz -83.48 deg; joints [7.258, -46.952, 74.618, -1.027, 57.231, -14.692, -89.958]
  MoveL 1126 to (-136.35, -13.61, 63.48) mm, rotated rx -114.61 ry 0 rz -83.29 deg; joints [7.394, -46.985, 74.719, -1.027, 57.241, -15.177, -90.224]
  MoveL 1127 to (-135.76, -14.07, 64.65) mm, rotated rx -114.97 ry 0 rz -83.12 deg; joints [7.484, -47.013, 74.788, -1.027, 57.251, -15.452, -90.447]
  MoveL 1128 to (-135.39, -14.51, 65.31) mm, rotated rx -114.97 ry 0 rz -83.12 deg; joints [7.507, -47.026, 74.788, -1.024, 57.29, -15.431, -90.473]
  MoveL 1129 to (-134.85, -16.26, 66.02) mm, rotated rx -114.97 ry 0 rz -83.12 deg; joints [7.534, -47.105, 74.788, -1.03, 57.347, -15.402, -90.449]
  MoveL 1130 to (-133.31, -26, 66.04) mm, rotated rx -114.98 ry 0 rz -78.96 deg; joints [7.536, -47.106, 74.79, -1.03, 57.347, -15.409, -94.61]
  MoveL 1131 to (-133.19, -26.82, 65.93) mm, rotated rx -114.96 ry 0 rz -78.81 deg; joints [7.53, -47.131, 74.787, -1.035, 57.347, -15.387, -94.729]
  MoveL 1132 to (-132.71, -29.77, 65.64) mm, rotated rx -114.82 ry 0 rz -77.47 deg; joints [7.501, -47.118, 74.769, -1.035, 57.336, -15.281, -96.055]
  MoveL 1133 to (-132.63, -30.55, 65.46) mm, rotated rx -114.79 ry 0 rz -77.38 deg; joints [7.492, -47.147, 74.764, -1.04, 57.336, -15.257, -96.116]
  MoveL 1134 to (-132.62, -32.3, 64.62) mm, rotated rx -114.39 ry 0 rz -76.3 deg; joints [7.407, -47.098, 74.716, -1.04, 57.289, -14.938, -97.152]
  MoveL 1135 to (-132.27, -33.65, 64.64) mm, rotated rx -114.39 ry 0 rz -75.71 deg; joints [7.409, -47.099, 74.717, -1.04, 57.289, -14.944, -97.739]
  MoveL 1136 to (-132.01, -34.95, 64.49) mm, rotated rx -114.34 ry 0 rz -75.32 deg; joints [7.397, -47.119, 74.71, -1.044, 57.289, -14.902, -98.098]
  MoveL 1137 to (-130.71, -42.04, 62.89) mm, rotated rx -113.68 ry 0 rz -71.97 deg; joints [7.25, -47.058, 74.619, -1.044, 57.235, -14.383, -101.367]
  MoveL 1138 to (-128.93, -45.38, 64.23) mm, rotated rx -114.29 ry 0 rz -70.23 deg; joints [7.38, -47.07, 74.719, -1.042, 57.236, -14.865, -103.2]
  MoveL 1139 to (-128.54, -46.25, 64.39) mm, rotated rx -114.29 ry 0 rz -70.23 deg; joints [7.387, -47.116, 74.719, -1.047, 57.255, -14.856, -103.173]
  MoveL 1140 to (-128.24, -47.09, 64.38) mm, rotated rx -114.28 ry 0 rz -69.85 deg; joints [7.385, -47.116, 74.718, -1.047, 57.255, -14.852, -103.546]
  MoveL 1141 to (-126.17, -53.24, 63.63) mm, rotated rx -113.98 ry 0 rz -67.26 deg; joints [7.319, -47.114, 74.668, -1.049, 57.255, -14.616, -106.095]
  MoveL 1142 to (-126.2, -53.19, 63.61) mm, rotated rx -114.54 ry 0 rz -66.19 deg; joints [7.389, -46.983, 74.71, -1.025, 57.255, -15.118, -107.34]
  MoveL 1143 to (-124.24, -53.95, 66.8) mm, rotated rx -115.89 ry 0 rz -65.55 deg; joints [7.683, -47.067, 74.949, -1.025, 57.263, -16.166, -108.134]
  MoveL 1144 to (-123.99, -54.03, 67.19) mm, rotated rx -116.06 ry 0 rz -65.47 deg; joints [7.72, -47.078, 74.981, -1.025, 57.263, -16.301, -108.232]
  MoveL 1145 to (-122.28, -54.76, 69.68) mm, rotated rx -117.48 ry 0 rz -64.81 deg; joints [7.999, -47.16, 75.231, -1.02, 57.263, -17.441, -109.062]
  MoveL 1146 to (-121.62, -54.01, 71.37) mm, rotated rx -118.38 ry 0 rz -64.99 deg; joints [8.181, -47.227, 75.403, -1.017, 57.263, -18.165, -108.983]
  MoveL 1147 to (-137.56, -61.45, 80.88) mm, rotated rx -118.38 ry 0 rz -64.99 deg; joints [8.432, -46.541, 73.647, -1.264, 57.263, -17.799, -107.891]
  Set speed (1000.0 mm/s)
  MoveL 1148 to (-122.96, -67.13, 98.06) mm, rotated rx -125.73 ry 0 rz -60.89 deg; joints [10.007, -47.264, 75.412, -1.203, 57.264, -23.598, -113.024]
  Set speed (5.0 mm/s)
  MoveL 1149 to (-108.78, -59.24, 86.38) mm, rotated rx -125.73 ry 0 rz -60.89 deg; joints [9.689, -47.953, 77.081, -0.941, 57.263, -24.041, -114.03]
  Set speed (16.7 mm/s)
  MoveL 1150 to (-109.6, -55.06, 88.11) mm, rotated rx -126.53 ry 0 rz -62.78 deg; joints [9.855, -48.038, 77.293, -0.924, 57.263, -24.683, -112.271]
  MoveL 1151 to (-109.69, -54.52, 88.34) mm, rotated rx -126.61 ry 0 rz -62.96 deg; joints [9.872, -48.04, 77.315, -0.92, 57.264, -24.742, -112.112]
  MoveL 1152 to (-110.14, -49.87, 90.49) mm, rotated rx -127.62 ry 0 rz -65.01 deg; joints [10.08, -48.152, 77.592, -0.895, 57.264, -25.556, -110.223]
  MoveL 1153 to (-110.47, -49.5, 90.29) mm, rotated rx -127.6 ry 0 rz -66.3 deg; joints [10.077, -48.273, 77.589, -0.926, 57.264, -25.526, -108.811]
  MoveL 1154 to (-110.74, -49.15, 90.15) mm, rotated rx -127.54 ry 0 rz -66.5 deg; joints [10.063, -48.266, 77.571, -0.927, 57.264, -25.474, -108.597]
  MoveL 1155 to (-113.2, -45.52, 89.01) mm, rotated rx -127.01 ry 0 rz -68.47 deg; joints [9.954, -48.199, 77.426, -0.938, 57.264, -25.056, -106.553]
  MoveL 1156 to (-113.75, -44.17, 88.98) mm, rotated rx -127.01 ry 0 rz -68.47 deg; joints [9.95, -48.125, 77.426, -0.924, 57.248, -25.067, -106.613]
  MoveL 1157 to (-113.85, -43.69, 89.08) mm, rotated rx -127.06 ry 0 rz -68.7 deg; joints [9.96, -48.13, 77.439, -0.922, 57.248, -25.108, -106.39]
  MoveL 1158 to (-113.83, -42.24, 89.81) mm, rotated rx -127.06 ry 0 rz -68.7 deg; joints [9.983, -48.069, 77.469, -0.902, 57.248, -25.094, -106.483]
  MoveL 1159 to (-112.96, -39.81, 91.98) mm, rotated rx -128.43 ry 0 rz -70.22 deg; joints [10.24, -48.28, 77.819, -0.887, 57.248, -26.208, -105.103]
  MoveL 1160 to (-113.22, -37.92, 92.45) mm, rotated rx -128.65 ry 0 rz -71.11 deg; joints [10.286, -48.307, 77.884, -0.88, 57.248, -26.392, -104.245]
  MoveL 1161 to (-113.16, -37.92, 92.52) mm, rotated rx -128.37 ry 0 rz -72.42 deg; joints [10.261, -48.444, 77.851, -0.921, 57.248, -26.117, -102.764]
  MoveL 1162 to (-115.33, -36.4, 90.45) mm, rotated rx -127.39 ry 0 rz -73.41 deg; joints [10.058, -48.329, 77.574, -0.945, 57.248, -25.32, -101.611]
  MoveL 1163 to (-116.24, -35.64, 89.58) mm, rotated rx -127.03 ry 0 rz -73.81 deg; joints [9.981, -48.279, 77.471, -0.952, 57.248, -25.043, -101.157]
  MoveL 1164 to (-117, -35.63, 88.59) mm, rotated rx -126.27 ry 0 rz -74.15 deg; joints [9.848, -48.237, 77.298, -0.973, 57.248, -24.4, -100.682]
  MoveL 1165 to (-117.3, -35.53, 88.23) mm, rotated rx -126.1 ry 0 rz -74.24 deg; joints [9.814, -48.219, 77.253, -0.977, 57.248, -24.266, -100.575]
  MoveL 1166 to (-118.82, -34.81, 86.45) mm, rotated rx -125.36 ry 0 rz -74.7 deg; joints [9.653, -48.131, 77.05, -0.991, 57.248, -23.68, -99.993]
  MoveL 1167 to (-119.06, -35.54, 85.84) mm, rotated rx -123.71 ry 0 rz -73.14 deg; joints [9.411, -47.887, 76.772, -0.991, 57.196, -22.273, -101.474]
  MoveL 1168 to (-118.72, -36.4, 85.95) mm, rotated rx -123.74 ry 0 rz -72.98 deg; joints [9.42, -47.91, 76.772, -0.992, 57.218, -22.293, -101.634]
  MoveL 1169 to (-117.63, -39.9, 85.89) mm, rotated rx -123.72 ry 0 rz -71.28 deg; joints [9.414, -47.908, 76.767, -0.992, 57.218, -22.273, -103.323]
  MoveL 1170 to (-117.55, -40.02, 85.95) mm, rotated rx -123.86 ry 0 rz -70.65 deg; joints [9.431, -47.847, 76.784, -0.976, 57.218, -22.405, -104.04]
  MoveL 1171 to (-116.07, -42, 87.01) mm, rotated rx -124.35 ry 0 rz -69.55 deg; joints [9.535, -47.897, 76.91, -0.967, 57.218, -22.8, -105.211]
  MoveL 1172 to (-115.72, -42.53, 87.22) mm, rotated rx -124.38 ry 0 rz -69.44 deg; joints [9.547, -47.916, 76.918, -0.967, 57.233, -22.819, -105.324]
  MoveL 1173 to (-114.38, -45.11, 87.69) mm, rotated rx -124.56 ry 0 rz -68.26 deg; joints [9.588, -47.955, 76.969, -0.967, 57.235, -22.96, -106.516]
  MoveL 1174 to (-113.68, -46.83, 87.7) mm, rotated rx -124.55 ry 0 rz -67.64 deg; joints [9.588, -47.983, 76.969, -0.973, 57.237, -22.945, -107.114]
  MoveL 1175 to (-110.62, -57.25, 85.4) mm, rotated rx -123.52 ry 0 rz -62.93 deg; joints [9.371, -47.911, 76.706, -0.998, 57.237, -22.117, -111.63]
  MoveL 1176 to (-109.2, -59.64, 85.56) mm, rotated rx -123.57 ry 0 rz -61.29 deg; joints [9.381, -47.872, 76.718, -0.988, 57.237, -22.159, -113.322]
  MoveL 1177 to (-109.19, -59.64, 85.56) mm, rotated rx -124.69 ry 0 rz -60.22 deg; joints [9.522, -47.811, 76.885, -0.947, 57.237, -23.163, -114.622]
  MoveL 1178 to (-108.79, -59.2, 86.38) mm, rotated rx -125.07 ry 0 rz -60.31 deg; joints [9.601, -47.85, 76.982, -0.94, 57.237, -23.465, -114.596]
  MoveL 1179 to (-123.01, -67.31, 97.87) mm, rotated rx -125.07 ry 0 rz -60.31 deg; joints [9.912, -47.16, 75.303, -1.202, 57.237, -23.029, -113.581]
  Set speed (1000.0 mm/s)
  MoveL 1180 to (-103.64, -86, 105.37) mm, rotated rx -128.85 ry 0 rz -50.56 deg; joints [10.675, -47.725, 76.329, -1.16, 57.237, -26.068, -123.783]
  Set speed (5.0 mm/s)
  MoveL 1181 to (-91.61, -76.1, 92.82) mm, rotated rx -128.85 ry 0 rz -50.56 deg; joints [10.329, -48.412, 77.952, -0.896, 57.237, -26.542, -124.747]
  Set speed (16.7 mm/s)
  MoveL 1182 to (-93.41, -74.47, 92.39) mm, rotated rx -128.64 ry 0 rz -51.71 deg; joints [10.286, -48.387, 77.889, -0.902, 57.237, -26.368, -123.558]
  MoveL 1183 to (-95.35, -73.29, 91.34) mm, rotated rx -128.03 ry 0 rz -53.07 deg; joints [10.172, -48.361, 77.732, -0.926, 57.237, -25.858, -122.066]
  MoveL 1184 to (-95.55, -73.36, 91.06) mm, rotated rx -126.5 ry 0 rz -53.42 deg; joints [9.969, -48.286, 77.461, -0.958, 57.237, -24.519, -121.524]
  MoveL 1185 to (-95.55, -74.38, 90.24) mm, rotated rx -126.11 ry 0 rz -53.03 deg; joints [9.888, -48.243, 77.354, -0.967, 57.237, -24.203, -121.848]
  MoveL 1186 to (-95.64, -74.93, 89.7) mm, rotated rx -126.11 ry 0 rz -53.03 deg; joints [9.869, -48.254, 77.33, -0.974, 57.237, -24.219, -121.813]
  MoveL 1187 to (-95.78, -75.25, 89.28) mm, rotated rx -126.04 ry 0 rz -53 deg; joints [9.845, -48.247, 77.299, -0.978, 57.237, -24.172, -121.821]
  MoveL 1188 to (-96.18, -75.88, 88.31) mm, rotated rx -125.59 ry 0 rz -52.87 deg; joints [9.751, -48.199, 77.179, -0.987, 57.237, -23.808, -121.873]
  MoveL 1189 to (-95.54, -78.96, 86.28) mm, rotated rx -124.14 ry 0 rz -51.2 deg; joints [9.487, -48.024, 76.848, -1.002, 57.237, -22.619, -123.39]
  MoveL 1190 to (-95.44, -79.45, 85.95) mm, rotated rx -124.04 ry 0 rz -51.06 deg; joints [9.462, -48.02, 76.819, -1.005, 57.237, -22.54, -123.505]
  MoveL 1191 to (-94.83, -82.94, 83.28) mm, rotated rx -122.81 ry 0 rz -49.64 deg; joints [9.204, -47.898, 76.513, -1.025, 57.237, -21.56, -124.737]
  MoveL 1192 to (-95.14, -84.13, 81.72) mm, rotated rx -122.81 ry 0 rz -49.64 deg; joints [9.15, -47.914, 76.453, -1.037, 57.237, -21.609, -124.661]
  MoveL 1193 to (-96.01, -84.33, 80.49) mm, rotated rx -122.72 ry 0 rz -49.65 deg; joints [9.094, -47.869, 76.39, -1.037, 57.232, -21.581, -124.634]
  MoveL 1194 to (-97.1, -84.13, 79.37) mm, rotated rx -122.23 ry 0 rz -50.03 deg; joints [8.988, -47.822, 76.272, -1.043, 57.232, -21.187, -124.182]
  MoveL 1195 to (-97.66, -84.48, 78.29) mm, rotated rx -121.34 ry 0 rz -50.24 deg; joints [8.834, -47.779, 76.105, -1.055, 57.232, -20.451, -123.846]
  MoveL 1196 to (-97.72, -84.46, 78.24) mm, rotated rx -120.36 ry 0 rz -49.67 deg; joints [8.701, -47.67, 75.979, -1.055, 57.193, -19.608, -124.361]
  MoveL 1197 to (-96.72, -86.5, 77.27) mm, rotated rx -119.93 ry 0 rz -48.7 deg; joints [8.608, -47.632, 75.881, -1.059, 57.193, -19.266, -125.276]
  MoveL 1198 to (-94.59, -89.92, 75.98) mm, rotated rx -119.32 ry 0 rz -46.83 deg; joints [8.479, -47.567, 75.748, -1.061, 57.193, -18.78, -127.073]
  MoveL 1199 to (-93.53, -90.67, 76.38) mm, rotated rx -119.49 ry 0 rz -45.54 deg; joints [8.512, -47.485, 75.775, -1.041, 57.192, -18.925, -128.479]
  MoveL 1200 to (-93.49, -90.71, 76.38) mm, rotated rx -120.86 ry 0 rz -44.91 deg; joints [8.692, -47.479, 75.958, -1.018, 57.193, -20.13, -129.291]
  MoveL 1201 to (-93.61, -86.15, 81.38) mm, rotated rx -123.07 ry 0 rz -46.39 deg; joints [9.163, -47.68, 76.477, -0.991, 57.193, -21.884, -128.129]
  MoveL 1202 to (-93.02, -85.01, 83.24) mm, rotated rx -124.19 ry 0 rz -46.87 deg; joints [9.377, -47.814, 76.731, -0.982, 57.193, -22.79, -127.773]
  MoveL 1203 to (-93.16, -83.79, 84.31) mm, rotated rx -124.24 ry 0 rz -46.95 deg; joints [9.421, -47.79, 76.782, -0.968, 57.193, -22.806, -127.768]
  MoveL 1204 to (-92.9, -82.93, 85.42) mm, rotated rx -124.75 ry 0 rz -47.15 deg; joints [9.527, -47.841, 76.912, -0.959, 57.193, -23.213, -127.64]
  MoveL 1205 to (-94.31, -77.17, 89.2) mm, rotated rx -126.91 ry 0 rz -49.91 deg; joints [9.944, -48.094, 77.445, -0.925, 57.193, -24.965, -125.161]
  MoveL 1206 to (-106.55, -87.47, 101.21) mm, rotated rx -126.91 ry 0 rz -49.91 deg; joints [10.272, -47.405, 75.792, -1.189, 57.193, -24.51, -124.169]
  Set speed (1000.0 mm/s)
  MoveL 1207 to (-103.93, -86.25, 104.91) mm, rotated rx -127.08 ry 0 rz -49.88 deg; joints [10.431, -47.526, 76.007, -1.181, 57.193, -24.524, -124.298]
  Set speed (5.0 mm/s)
  MoveL 1208 to (-91.73, -75.97, 92.86) mm, rotated rx -127.08 ry 0 rz -49.88 deg; joints [10.102, -48.217, 77.657, -0.915, 57.193, -24.981, -125.283]
  Set speed (16.7 mm/s)
  MoveL 1209 to (-103.58, -86.48, 105.05) mm, rotated rx -127.14 ry 0 rz -49.71 deg; joints [10.444, -47.533, 76.025, -1.179, 57.193, -24.573, -124.481]
  Set speed (1000.0 mm/s)
  MoveL 1210 to (19.02, -119.65, 120.7) mm, rotated rx -135.48 ry 0 rz 8.18 deg; joints [12.257, -50.655, 80.58, -2.101, 53.502, -30.552, -180]
  Set speed (5.0 mm/s)
  MoveL 1211 to (17.02, -105.77, 106.44) mm, rotated rx -135.48 ry 0 rz 8.18 deg; joints [11.892, -51.74, 82.526, -2.072, 52.631, -30.907, -180]
  Set speed (16.7 mm/s)
  MoveL 1212 to (14.76, -107.9, 104.63) mm, rotated rx -134.52 ry 0 rz 6.86 deg; joints [11.704, -51.618, 82.224, -2.096, 52.631, -30.129, -178.495]
  MoveL 1213 to (14.43, -108.18, 104.38) mm, rotated rx -134.41 ry 0 rz 6.69 deg; joints [11.681, -51.6, 82.187, -2.098, 52.631, -30.041, -178.313]
  MoveL 1214 to (12.82, -109.35, 103.37) mm, rotated rx -133.94 ry 0 rz 5.87 deg; joints [11.582, -51.529, 82.031, -2.108, 52.631, -29.659, -177.404]
  MoveL 1215 to (10.78, -109.96, 102.95) mm, rotated rx -133.95 ry 0 rz 5.83 deg; joints [11.564, -51.442, 82.031, -2.104, 52.554, -29.691, -177.379]
  MoveL 1216 to (9.53, -109.72, 103.33) mm, rotated rx -133.96 ry 0 rz 5.81 deg; joints [11.576, -51.382, 82.045, -2.084, 52.554, -29.698, -177.432]
  MoveL 1217 to (8.48, -108.78, 104.41) mm, rotated rx -133.97 ry 0 rz 5.78 deg; joints [11.617, -51.358, 82.106, -2.066, 52.554, -29.679, -177.489]
  MoveL 1218 to (8.74, -107.31, 105.9) mm, rotated rx -133.99 ry 0 rz 5.75 deg; joints [11.679, -51.422, 82.204, -2.065, 52.556, -29.632, -177.489]
  MoveL 1219 to (9.83, -105.96, 107.16) mm, rotated rx -134.67 ry 0 rz 6.41 deg; joints [11.811, -51.507, 82.416, -2.048, 52.556, -30.184, -178.277]
  MoveL 1220 to (10.74, -103.69, 109.27) mm, rotated rx -136.02 ry 0 rz 7.2 deg; joints [12.059, -51.657, 82.823, -2.007, 52.556, -31.306, -179.323]
  MoveL 1221 to (10.56, -101.91, 110.95) mm, rotated rx -137.24 ry 0 rz 7.31 deg; joints [12.273, -51.799, 83.189, -1.97, 52.556, -32.335, -179.662]
  MoveL 1222 to (12.28, -115.38, 125.63) mm, rotated rx -137.24 ry 0 rz 7.31 deg; joints [12.698, -51.169, 81.754, -2.287, 52.556, -31.745, -178.816]
  Set speed (1000.0 mm/s)
  MoveL 1223 to (17.45, -114.14, 126.15) mm, rotated rx -137.29 ry 0 rz 7.51 deg; joints [12.734, -51.385, 81.754, -2.302, 52.727, -31.754, -178.963]
  Set speed (5.0 mm/s)
  MoveL 1224 to (15.68, -100.69, 111.46) mm, rotated rx -137.29 ry 0 rz 7.51 deg; joints [12.308, -52.016, 83.184, -1.986, 52.727, -32.344, -179.804]
  Set speed (16.7 mm/s)
  MoveL 1225 to (17.4, -103.52, 108.57) mm, rotated rx -135.68 ry 0 rz 8.24 deg; joints [12.011, -51.918, 82.787, -2.111, 52.493, -30.966, -180]
  MoveL 1226 to (19.41, -117.35, 122.88) mm, rotated rx -135.68 ry 0 rz 8.24 deg; joints [12.423, -51.289, 81.336, -2.432, 52.493, -30.387, -179.135]
  Set speed (1000.0 mm/s)
  MoveL 1227 to (111.82, -88.61, 94.29) mm, rotated rx -124.07 ry 0 rz 52.29 deg; joints [12.529, -72.362, 105.206, -57.309, 12.995, 31.469, -180]
  Set speed (5.0 mm/s)
  MoveL 1228 to (98.71, -78.48, 83.09) mm, rotated rx -124.07 ry 0 rz 52.29 deg; joints [12.178, -72.815, 106.773, -61.116, 12.173, 35.172, -180]
  Set speed (16.7 mm/s)
  MoveL 1229 to (95.71, -79.78, 85.34) mm, rotated rx -125.1 ry 0 rz 50.98 deg; joints [12.426, -72.684, 106.821, -61.121, 12.349, 34.342, -178.921]
  MoveL 1230 to (94.31, -79.63, 87.01) mm, rotated rx -125.1 ry 0 rz 50.98 deg; joints [12.489, -72.592, 106.799, -61.121, 12.39, 34.395, -179.003]
  MoveL 1231 to (93.97, -78.83, 88.11) mm, rotated rx -125.19 ry 0 rz 50.99 deg; joints [12.553, -72.592, 106.836, -61.159, 12.434, 34.391, -179.057]
  MoveL 1232 to (93.9, -77.73, 89.14) mm, rotated rx -125.67 ry 0 rz 51.37 deg; joints [12.675, -72.565, 106.913, -61.556, 12.485, 34.39, -179.477]
  MoveL 1233 to (93.88, -77.81, 89.09) mm, rotated rx -126.51 ry 0 rz 51.44 deg; joints [12.806, -72.55, 107.028, -62.301, 12.513, 34.389, -179.528]
  MoveL 1234 to (92.11, -77.64, 91.07) mm, rotated rx -127.44 ry 0 rz 50.98 deg; joints [13.026, -72.434, 107.087, -62.301, 12.664, 33.631, -179.286]
  MoveL 1235 to (91.71, -77.52, 91.58) mm, rotated rx -127.44 ry 0 rz 50.98 deg; joints [13.046, -72.411, 107.086, -62.301, 12.677, 33.648, -179.311]
  MoveL 1236 to (91.21, -76.9, 92.59) mm, rotated rx -127.46 ry 0 rz 50.98 deg; joints [13.094, -72.399, 107.107, -62.301, 12.71, 33.661, -179.351]
  MoveL 1237 to (91.08, -75.99, 93.47) mm, rotated rx -127.6 ry 0 rz 51.04 deg; joints [13.156, -72.404, 107.148, -62.301, 12.754, 33.572, -179.469]
  MoveL 1238 to (91.83, -74.28, 94.11) mm, rotated rx -127.6 ry 0 rz 51.04 deg; joints [13.2, -72.519, 107.242, -62.276, 12.795, 33.572, -179.468]
  MoveL 1239 to (92.82, -73.23, 93.96) mm, rotated rx -127.6 ry 0 rz 51.26 deg; joints [13.204, -72.593, 107.289, -62.276, 12.803, 33.567, -179.661]
  MoveL 1240 to (98.07, -69, 91.8) mm, rotated rx -126.56 ry 0 rz 54.42 deg; joints [13.179, -73.868, 108.951, -76.759, 12.069, 48.815, -180]
  MoveL 1241 to (98.89, -68.19, 91.53) mm, rotated rx -126.5 ry 0 rz 54.78 deg; joints [13.191, -74.054, 109.192, -78.754, 12.045, 50.844, -180]
  MoveL 1242 to (101.69, -66.18, 89.92) mm, rotated rx -125.74 ry 0 rz 56.33 deg; joints [13.126, -74.756, 110.076, -87.018, 12.006, 59.693, -180]
  MoveL 1243 to (103.03, -65.73, 88.72) mm, rotated rx -125.71 ry 0 rz 56.31 deg; joints [13.082, -74.869, 110.122, -87.019, 11.98, 59.679, -179.92]
  MoveL 1244 to (103.68, -66.1, 87.68) mm, rotated rx -125.69 ry 0 rz 56.3 deg; joints [13.035, -74.9, 110.114, -87.037, 11.947, 59.679, -179.87]
  MoveL 1245 to (103.76, -67.85, 86.24) mm, rotated rx -125.66 ry 0 rz 56.28 deg; joints [12.953, -74.834, 110.021, -87.059, 11.884, 59.679, -179.824]
  MoveL 1246 to (103.3, -69.35, 85.59) mm, rotated rx -125.36 ry 0 rz 55.58 deg; joints [12.879, -74.87, 109.998, -87.059, 11.831, 59.924, -179.079]
  MoveL 1247 to (103.11, -71.12, 84.37) mm, rotated rx -124.67 ry 0 rz 54.64 deg; joints [12.723, -74.985, 109.979, -87.058, 11.722, 60.5, -178.014]
  MoveL 1248 to (116.52, -80.64, 95.75) mm, rotated rx -124.67 ry 0 rz 54.64 deg; joints [13.179, -75.044, 109.13, -86.99, 12.227, 60.502, -177.103]
  Set speed (1000.0 mm/s)
  MoveL 1249 to (114.8, -107.23, 67.61) mm, rotated rx -113.91 ry 0 rz 47.56 deg; joints [10.184, -76.163, 108.45, -86.989, 9.933, 69.279, -168.44]
  Set speed (5.0 mm/s)
  MoveL 1250 to (101.3, -94.89, 59.5) mm, rotated rx -113.91 ry 0 rz 47.56 deg; joints [9.85, -75.972, 109.258, -86.999, 9.544, 69.277, -169.44]
  Set speed (16.7 mm/s)
  MoveL 1251 to (98.73, -96.19, 61.7) mm, rotated rx -114.82 ry 0 rz 46.44 deg; joints [10.1, -75.873, 109.285, -86.999, 9.74, 68.527, -168.436]
  MoveL 1252 to (98.26, -96.39, 62.13) mm, rotated rx -114.95 ry 0 rz 46.3 deg; joints [10.14, -75.848, 109.285, -87.031, 9.771, 68.456, -168.316]
  MoveL 1253 to (95.88, -97.29, 64.41) mm, rotated rx -115.89 ry 0 rz 45.36 deg; joints [10.397, -75.742, 109.315, -87.031, 9.97, 67.686, -167.493]
  MoveL 1254 to (94.8, -97.08, 66.3) mm, rotated rx -115.89 ry 0 rz 45.36 deg; joints [10.473, -75.663, 109.292, -87.031, 10.027, 67.738, -167.544]
  MoveL 1255 to (94.8, -96.05, 67.78) mm, rotated rx -116.01 ry 0 rz 45.38 deg; joints [10.564, -75.679, 109.342, -87.031, 10.099, 67.673, -167.595]
  MoveL 1256 to (95.87, -92.99, 70.48) mm, rotated rx -117.16 ry 0 rz 46.64 deg; joints [10.874, -75.549, 109.388, -87.032, 10.338, 66.72, -169.012]
  MoveL 1257 to (96.02, -92.6, 70.8) mm, rotated rx -117.27 ry 0 rz 46.77 deg; joints [10.906, -75.542, 109.398, -87.032, 10.362, 66.637, -169.153]
  MoveL 1258 to (97.67, -89.01, 73.11) mm, rotated rx -118.18 ry 0 rz 48.27 deg; joints [11.16, -75.456, 109.457, -87.032, 10.556, 65.897, -170.779]
  MoveL 1259 to (98.21, -88.1, 73.48) mm, rotated rx -118.18 ry 0 rz 48.27 deg; joints [11.185, -75.526, 109.517, -87.02, 10.578, 65.897, -170.769]
  MoveL 1260 to (98.6, -87.61, 73.56) mm, rotated rx -118.21 ry 0 rz 48.54 deg; joints [11.195, -75.522, 109.518, -87.02, 10.586, 65.867, -171.045]
  MoveL 1261 to (101.35, -84.17, 73.8) mm, rotated rx -118.31 ry 0 rz 50.36 deg; joints [11.224, -75.527, 109.536, -87.021, 10.608, 65.787, -172.873]
  MoveL 1262 to (101.34, -84.09, 73.92) mm, rotated rx -118.79 ry 0 rz 51.22 deg; joints [11.295, -75.375, 109.488, -87.447, 10.66, 65.787, -173.758]
  MoveL 1263 to (101.4, -82.67, 75.44) mm, rotated rx -119.45 ry 0 rz 51.72 deg; joints [11.47, -75.298, 109.521, -87.447, 10.792, 65.241, -174.354]
  MoveL 1264 to (101.61, -81.77, 76.13) mm, rotated rx -119.45 ry 0 rz 51.72 deg; joints [11.507, -75.346, 109.572, -87.425, 10.823, 65.241, -174.358]
  MoveL 1265 to (102.31, -80.38, 76.63) mm, rotated rx -120.21 ry 0 rz 52.89 deg; joints [11.645, -75.218, 109.571, -87.721, 10.926, 64.877, -175.587]
  MoveL 1266 to (101.66, -78.53, 79.4) mm, rotated rx -121.97 ry 0 rz 53.39 deg; joints [12.049, -75.031, 109.66, -87.721, 11.226, 63.391, -176.325]
  MoveL 1267 to (99.3, -78.11, 82.72) mm, rotated rx -123.47 ry 0 rz 52.9 deg; joints [12.43, -74.853, 109.757, -87.722, 11.505, 62.168, -176.08]
  MoveL 1268 to (112.61, -88.17, 93.75) mm, rotated rx -123.47 ry 0 rz 52.9 deg; joints [12.873, -74.932, 108.914, -87.66, 11.998, 62.169, -175.15]
  Set speed (1000.0 mm/s)
  MoveL 1269 to (116.23, -82.13, 94.81) mm, rotated rx -123.04 ry 0 rz 54.09 deg; joints [12.889, -75.211, 109.085, -87.238, 12.018, 62.169, -176.317]
  Set speed (5.0 mm/s)
  MoveL 1270 to (102.65, -72.3, 83.9) mm, rotated rx -123.04 ry 0 rz 54.09 deg; joints [12.45, -75.133, 109.93, -87.295, 11.528, 62.167, -177.246]
  Set speed (16.7 mm/s)
  MoveL 1271 to (106.23, -70.25, 81.17) mm, rotated rx -121.79 ry 0 rz 55.79 deg; joints [12.132, -75.281, 109.849, -87.295, 11.295, 63.188, -178.74]
  MoveL 1272 to (107.41, -70.03, 79.78) mm, rotated rx -121.79 ry 0 rz 55.79 deg; joints [12.081, -75.373, 109.883, -87.295, 11.26, 63.147, -178.687]
  MoveL 1273 to (107.81, -70.26, 79.04) mm, rotated rx -121.68 ry 0 rz 55.8 deg; joints [12.031, -75.395, 109.871, -87.295, 11.224, 63.222, -178.67]
  MoveL 1274 to (108.44, -71.07, 77.43) mm, rotated rx -120.43 ry 0 rz 55.77 deg; joints [11.755, -75.502, 109.797, -87.295, 11.018, 64.292, -178.482]
  MoveL 1275 to (109.35, -70.9, 76.31) mm, rotated rx -119.93 ry 0 rz 56.06 deg; joints [11.626, -75.56, 109.77, -87.294, 10.921, 64.697, -178.693]
  MoveL 1276 to (109.83, -70.87, 75.65) mm, rotated rx -119.74 ry 0 rz 56.14 deg; joints [11.567, -75.596, 109.765, -87.295, 10.877, 64.848, -178.736]
  MoveL 1277 to (112.42, -70.9, 71.71) mm, rotated rx -118.07 ry 0 rz 56.73 deg; joints [11.121, -75.794, 109.684, -87.294, 10.54, 66.22, -179.09]
  MoveL 1278 to (112.82, -71.03, 70.95) mm, rotated rx -118.07 ry 0 rz 56.73 deg; joints [11.088, -75.817, 109.685, -87.294, 10.516, 66.198, -179.071]
  MoveL 1279 to (113.05, -72.18, 69.4) mm, rotated rx -118.07 ry 0 rz 56.73 deg; joints [11.014, -75.785, 109.631, -87.34, 10.457, 66.197, -179.045]
  MoveL 1280 to (112.93, -72.8, 68.95) mm, rotated rx -117.88 ry 0 rz 56.49 deg; joints [10.963, -75.807, 109.623, -87.34, 10.418, 66.354, -178.773]
  MoveL 1281 to (112.56, -73.82, 68.46) mm, rotated rx -117.88 ry 0 rz 56.49 deg; joints [10.932, -75.737, 109.561, -87.356, 10.391, 66.354, -178.781]
  MoveL 1282 to (109.25, -79.9, 66.98) mm, rotated rx -117.25 ry 0 rz 53.57 deg; joints [10.763, -75.808, 109.535, -87.356, 10.262, 66.87, -175.777]
  MoveL 1283 to (108.79, -81.97, 65.21) mm, rotated rx -116.26 ry 0 rz 52.26 deg; joints [10.527, -75.976, 109.535, -87.058, 10.081, 67.409, -174.371]
  MoveL 1284 to (108.14, -83.32, 64.58) mm, rotated rx -116.26 ry 0 rz 52.26 deg; joints [10.487, -75.878, 109.45, -87.079, 10.046, 67.409, -174.383]
  MoveL 1285 to (107.3, -84.35, 64.64) mm, rotated rx -116.25 ry 0 rz 52.15 deg; joints [10.478, -75.798, 109.391, -87.078, 10.036, 67.42, -174.287]
  MoveL 1286 to (106.13, -85.42, 65.16) mm, rotated rx -116.5 ry 0 rz 51 deg; joints [10.554, -75.859, 109.465, -87.079, 10.098, 67.211, -173.153]
  MoveL 1287 to (103.81, -89.56, 63.3) mm, rotated rx -115.13 ry 0 rz 48.24 deg; joints [10.251, -76.085, 109.465, -86.386, 9.863, 67.696, -170.301]
  MoveL 1288 to (103.98, -91.37, 60.39) mm, rotated rx -113.92 ry 0 rz 47.73 deg; joints [9.918, -76.217, 109.428, -86.386, 9.604, 68.694, -169.636]
  MoveL 1289 to (117.51, -103.67, 68.5) mm, rotated rx -113.92 ry 0 rz 47.73 deg; joints [10.252, -76.403, 108.617, -86.374, 9.992, 68.694, -168.643]
  Set speed (1000.0 mm/s)
  MoveL 1290 to (138.84, -95.44, -29.33) mm, rotated rx -80.82 ry 0 rz 55.97 deg; joints [-0.164, -77.905, 108.789, -58.872, 1.397, 68.695, -176.192]
  Set speed (5.0 mm/s)
  MoveL 1291 to (122.47, -84.4, -26.14) mm, rotated rx -80.82 ry 0 rz 55.97 deg; joints [-0.025, -77.539, 109.482, -58.871, 1.519, 68.792, -177.311]
  Set speed (16.7 mm/s)
  MoveL 1292 to (121.83, -85.61, -25.22) mm, rotated rx -81.17 ry 0 rz 55.45 deg; joints [0.082, -77.523, 109.436, -59.169, 1.618, 68.792, -176.799]
  MoveL 1293 to (121.51, -86.3, -24.42) mm, rotated rx -81.17 ry 0 rz 55.45 deg; joints [0.116, -77.458, 109.376, -59.168, 1.651, 68.81, -176.82]
  MoveL 1294 to (121.4, -86.6, -23.89) mm, rotated rx -81.37 ry 0 rz 55.33 deg; joints [0.177, -77.448, 109.35, -59.338, 1.708, 68.809, -176.708]
  MoveL 1295 to (121.32, -86.89, -23.19) mm, rotated rx -81.37 ry 0 rz 55.33 deg; joints [0.207, -77.42, 109.319, -59.338, 1.737, 68.825, -176.719]
  MoveL 1296 to (121.66, -86.85, -21.5) mm, rotated rx -81.37 ry 0 rz 55.33 deg; joints [0.281, -77.423, 109.297, -59.338, 1.809, 68.865, -176.73]
  MoveL 1297 to (123.29, -85.43, -17.57) mm, rotated rx -82.88 ry 0 rz 56.12 deg; joints [0.734, -77.353, 109.118, -60.598, 2.222, 68.865, -177.581]
  MoveL 1298 to (123.63, -85.07, -16.92) mm, rotated rx -82.88 ry 0 rz 56.12 deg; joints [0.763, -77.385, 109.134, -60.583, 2.251, 68.865, -177.578]
  MoveL 1299 to (124.64, -83.71, -16.25) mm, rotated rx -82.88 ry 0 rz 56.12 deg; joints [0.796, -77.509, 109.216, -60.567, 2.283, 68.865, -177.552]
  MoveL 1300 to (124.99, -83.19, -16.24) mm, rotated rx -82.88 ry 0 rz 56.37 deg; joints [0.796, -77.509, 109.216, -60.569, 2.284, 68.865, -177.794]
  MoveL 1301 to (125.61, -82.2, -16.51) mm, rotated rx -82.88 ry 0 rz 56.37 deg; joints [0.787, -77.601, 109.287, -60.569, 2.275, 68.859, -177.769]
  MoveL 1302 to (128.29, -77.31, -19.31) mm, rotated rx -81.81 ry 0 rz 58.49 deg; joints [0.463, -77.652, 109.412, -59.673, 1.982, 68.859, -179.86]
  MoveL 1303 to (128.77, -76.11, -20.82) mm, rotated rx -81.81 ry 0 rz 58.49 deg; joints [0.399, -77.763, 109.516, -59.673, 1.92, 68.825, -179.822]
  MoveL 1304 to (128.6, -75.88, -22.52) mm, rotated rx -80.71 ry 0 rz 58.83 deg; joints [0.118, -77.821, 109.691, -64.035, 1.582, 74.14, -180]
  MoveL 1305 to (129, -74.93, -23.4) mm, rotated rx -80.37 ry 0 rz 59.22 deg; joints [0.02, -78.041, 110.021, -82.03, 1.358, 92.416, -180]
  MoveL 1306 to (129.03, -74.88, -23.37) mm, rotated rx -78.87 ry -29.53 rz 54.89 deg; joints [7.318, -78.435, 111.32, -91.862, 37.251, 108.689, -172.1]
  MoveL 1307 to (130.64, -72.67, -21.45) mm, rotated rx -81.07 ry 0 rz 61.47 deg; joints [0.261, -79.003, 111.495, -148.389, 3.02, 158.184, -180]
  MoveL 1308 to (131.06, -72.02, -21.04) mm, rotated rx -81.13 ry 0 rz 61.62 deg; joints [0.293, -79.102, 111.61, -149.406, 3.171, 159.151, -180]
  MoveL 1309 to (133.41, -67.9, -19.93) mm, rotated rx -81.49 ry 0 rz 63.24 deg; joints [0.435, -79.966, 112.808, -159.372, 5.003, 168.81, -180]
  MoveL 1310 to (133.8, -67.15, -19.89) mm, rotated rx -81.49 ry 0 rz 63.24 deg; joints [0.438, -80.035, 112.864, -159.371, 5.013, 168.81, -179.978]
  MoveL 1311 to (134.25, -66.19, -20.09) mm, rotated rx -81.47 ry 0 rz 63.4 deg; joints [0.428, -80.153, 113.005, -160.1, 5.168, 169.552, -180]
  MoveL 1312 to (135.7, -62.67, -21.57) mm, rotated rx -80.91 ry 0 rz 64.86 deg; joints [0.269, -80.902, 114.146, -166.265, 6.907, 176.187, -180]
  MoveL 1313 to (137.15, -59.17, -22.28) mm, rotated rx -80.59 ry 0 rz 66.48 deg; joints [0.193, -81.683, 115.366, -169.709, 8.918, 179.898, -180]
  MoveL 1314 to (137.34, -58.68, -22.4) mm, rotated rx -80.55 ry 0 rz 66.63 deg; joints [0.182, -81.765, 115.485, -169.965, 9.097, 180.184, -180]
  MoveL 1315 to (138.52, -55.33, -23.62) mm, rotated rx -80.11 ry 0 rz 67.91 deg; joints [0.052, -82.405, 116.488, -172.042, 10.702, 182.629, -180]
  MoveL 1316 to (138.88, -54.28, -23.91) mm, rotated rx -79.98 ry 0 rz 68.4 deg; joints [0.016, -82.629, 116.857, -172.622, 11.329, 183.321, -180]
  MoveL 1317 to (141.71, -44.3, -27.64) mm, rotated rx -78.56 ry 0 rz 72.31 deg; joints [-0.413, -84.446, 119.895, -176.199, 16.406, 188.083, -180]
  MoveL 1318 to (141.88, -43.31, -28.3) mm, rotated rx -78.56 ry 0 rz 72.31 deg; joints [-0.444, -84.516, 119.957, -176.3, 16.397, 188.17, -180]
  MoveL 1319 to (141.91, -42.89, -28.8) mm, rotated rx -78.49 ry 0 rz 72.37 deg; joints [-0.481, -84.562, 120.03, -176.445, 16.486, 188.367, -180]
  MoveL 1320 to (141.9, -41.96, -30.15) mm, rotated rx -77.64 ry 0 rz 73.08 deg; joints [-0.719, -84.801, 120.571, -177.384, 17.489, 190.047, -180]
  MoveL 1321 to (142.62, -37.71, -32.31) mm, rotated rx -76.8 ry 0 rz 74.75 deg; joints [-0.991, -85.499, 121.87, -178.429, 19.742, 191.796, -180]
  MoveL 1322 to (142.69, -36.46, -33.43) mm, rotated rx -76.31 ry 0 rz 74.72 deg; joints [-1.149, -85.573, 121.971, -178.879, 19.742, 192.674, -180]
  MoveL 1323 to (142.55, -36.21, -34.26) mm, rotated rx -76.05 ry 0 rz 74.71 deg; joints [-1.243, -85.58, 122.004, -179.146, 19.753, 193.153, -180]
  MoveL 1324 to (141.72, -37.09, -36.6) mm, rotated rx -75.28 ry 0 rz 74.67 deg; joints [-1.52, -85.478, 122.006, -179.931, 19.815, 194.587, -180]
  MoveL 1325 to (141.78, -34.82, -38.6) mm, rotated rx -74.5 ry 0 rz 75.53 deg; joints [-1.782, -85.811, 122.714, -180.64, 21.054, 195.958, -180]
  MoveL 1326 to (141.86, -33.98, -39.09) mm, rotated rx -74.35 ry 0 rz 75.82 deg; joints [-1.838, -85.93, 122.946, -180.778, 21.457, 196.222, -180]
  MoveL 1327 to (141.57, -29.29, -43.66) mm, rotated rx -72.55 ry 0 rz 77.59 deg; joints [-2.451, -86.549, 124.414, -182.167, 24.087, 199.137, -180]
  MoveL 1328 to (141.21, -28.39, -45.4) mm, rotated rx -72.53 ry 0 rz 77.55 deg; joints [-2.544, -86.592, 124.479, -182.388, 24.087, 199.337, -179.99]
  MoveL 1329 to (140.47, -29.16, -47.19) mm, rotated rx -72.51 ry 0 rz 77.52 deg; joints [-2.637, -86.507, 124.436, -182.609, 24.097, 199.536, -179.99]
  MoveL 1330 to (139.72, -31.68, -47.77) mm, rotated rx -72.48 ry 0 rz 77.47 deg; joints [-2.67, -86.308, 124.274, -182.685, 24.097, 199.624, -179.982]
  MoveL 1331 to (139.19, -35.08, -46.94) mm, rotated rx -72.81 ry 0 rz 76.1 deg; joints [-2.559, -86.339, 124.267, -182.421, 24.097, 199.079, -178.569]
  MoveL 1332 to (139.1, -35.47, -46.89) mm, rotated rx -72.85 ry 0 rz 75.86 deg; joints [-2.549, -86.351, 124.268, -182.401, 24.075, 199.028, -178.337]
  MoveL 1333 to (138.15, -39.86, -46.17) mm, rotated rx -73.13 ry 0 rz 74.07 deg; joints [-2.453, -86.376, 124.262, -182.173, 24.075, 198.557, -176.514]
